LIN {X 0,Y 218.503,Z 629.529,A -85,B 0,C 180,E1 -20253.691,E2 -20253.691} C_VEL
LIN {X 0,Y 218.752,Z 627.483,A -85,B 0,C 180,E1 -20257.386,E2 -20257.386} C_VEL
LIN {X 0,Y 219.498,Z 624.035,A -85,B 0,C 180,E1 -20261.078,E2 -20261.078} C_VEL
LIN {X 0,Y 220.889,Z 619.081,A -85,B 0,C 180,E1 -20264.748,E2 -20264.748} C_VEL
LIN {X 0,Y 221.921,Z 616.025,A -85,B 0,C 180,E1 -20266.562,E2 -20266.562} C_VEL
LIN {X 0,Y 224.966,Z 612.775,A -85,B 0,C 180,E1 -20270.412,E2 -20270.412} C_VEL
LIN {X 0,Y 228.61,Z 608.967,A -85,B 0,C 180,E1 -20273.558,E2 -20273.558} C_VEL
LIN {X 0,Y 233.431,Z 603.675,A -85,B 0,C 180,E1 -20276.849,E2 -20276.849} C_VEL
LIN {X 0,Y 239.262,Z 597.121,A -85,B 0,C 180,E1 -20279.959,E2 -20279.959} C_VEL
LIN {X 0,Y 246.121,Z 589.152,A -85,B 0,C 180,E1 -20282.859,E2 -20282.859} C_VEL
LIN {X 0,Y 253.842,Z 579.668,A -85,B 0,C 180,E1 -20285.552,E2 -20285.552} C_VEL
LIN {X 0,Y 259.519,Z 572.234,A -85,B 0,C 180,E1 -20287.233,E2 -20287.233} C_VEL
LIN {X 0,Y 261.796,Z 567.859,A -85,B 0,C 180,E1 -20288.621,E2 -20288.621} C_VEL
LIN {X 0,Y 263.848,Z 563.319,A -85,B 0,C 180,E1 -20290.262,E2 -20290.262} C_VEL
LIN {X 0,Y 264.397,Z 560.907,A -85,B 0,C 180,E1 -20291.648,E2 -20291.648} C_VEL
LIN {X 0,Y 264.273,Z 558.69,A -85,B 0,C 180,E1 -20294.108,E2 -20294.108} C_VEL
LIN {X 0,Y 264.108,Z 557.741,A -85,B 0,C 180,E1 -20296.222,E2 -20296.222} C_VEL
LIN {X 0,Y 263.97,Z 557.685,A -85,B 0,C 180,E1 -20298.271,E2 -20298.271} C_VEL
LIN {X 0,Y 263.62,Z 558.789,A -85,B 0,C 180,E1 -20300.638,E2 -20300.638} C_VEL
LIN {X 0,Y 263.042,Z 560.356,A -85,B 0,C 180,E1 -20302.083,E2 -20302.083} C_VEL
LIN {X 0,Y 261.574,Z 564.149,A -85,B 0,C 180,E1 -20304.563,E2 -20304.563} C_VEL
LIN {X 0,Y 260.042,Z 567.586,A -85,B 0,C 180,E1 -20306.355,E2 -20306.355} C_VEL
LIN {X 0,Y 252.229,Z 576.861,A -85,B 0,C 180,E1 -20308.971,E2 -20308.971} C_VEL
LIN {X 0,Y 245.081,Z 584.507,A -85,B 0,C 180,E1 -20311.761,E2 -20311.761} C_VEL
LIN {X 0,Y 238.602,Z 590.64,A -85,B 0,C 180,E1 -20314.717,E2 -20314.717} C_VEL
LIN {X 0,Y 233.176,Z 595.264,A -85,B 0,C 180,E1 -20317.867,E2 -20317.867} C_VEL
LIN {X 0,Y 229.685,Z 597.919,A -85,B 0,C 180,E1 -20320.331,E2 -20320.331} C_VEL
LIN {X 0,Y 225.704,Z 600.243,A -85,B 0,C 180,E1 -20323.725,E2 -20323.725} C_VEL
LIN {X 0,Y 222.922,Z 601.265,A -85,B 0,C 180,E1 -20327.251,E2 -20327.251} C_VEL
LIN {X 0,Y 220.73,Z 600.99,A -85,B 0,C 180,E1 -20330.84,E2 -20330.84} C_VEL
LIN {X 0,Y 219.454,Z 599.351,A -85,B 0,C 180,E1 -20334.487,E2 -20334.487} C_VEL
LIN {X 0,Y 218.949,Z 596.268,A -85,B 0,C 180,E1 -20338.161,E2 -20338.161} C_VEL
LIN {X 0,Y 218.827,Z 591.637,A -85,B 0,C 180,E1 -20341.841,E2 -20341.841} C_VEL
LIN {X 0,Y 218.85,Z 586.867,A -85,B 0,C 180,E1 -20344.699,E2 -20344.699} C_VEL
LIN {X 0,Y 219.289,Z 580.046,A -85,B 0,C 180,E1 -20347.932,E2 -20347.932} C_VEL
LIN {X 0,Y 220.063,Z 571.783,A -85,B 0,C 180,E1 -20351.047,E2 -20351.047} C_VEL
LIN {X 0,Y 221.026,Z 562.858,A -85,B 0,C 180,E1 -20353.797,E2 -20353.797} C_VEL
LIN {X 0,Y 222.231,Z 554.062,A -85,B 0,C 180,E1 -20356.065,E2 -20356.065} C_VEL
LIN {X 0,Y 223.678,Z 543.655,A -85,B 0,C 180,E1 -20358.313,E2 -20358.313} C_VEL
LIN {X 0,Y 225.283,Z 531.049,A -85,B 0,C 180,E1 -20360.519,E2 -20360.519} C_VEL
LIN {X 0,Y 225.813,Z 526.308,A -85,B 0,C 180,E1 -20361.239,E2 -20361.239} C_VEL
LIN {X 0,Y 223.814,Z 512.351,A -85,B 0,C 180,E1 -20363.186,E2 -20363.186} C_VEL
LIN {X 0,Y 221.525,Z 497.373,A -85,B 0,C 180,E1 -20364.871,E2 -20364.871} C_VEL
LIN {X 0,Y 219.985,Z 485.91,A -85,B 0,C 180,E1 -20365.931,E2 -20365.931} C_VEL
LIN {X 0,Y 220.619,Z 480.954,A -85,B 0,C 180,E1 -20370.668,E2 -20370.668} C_VEL
LIN {X 0,Y 221.078,Z 477.085,A -85,B 0,C 180,E1 -20374.453,E2 -20374.453} C_VEL
LIN {X 0,Y 221.122,Z 476.819,A -85,B 0,C 180,E1 -20374.897,E2 -20374.897} C_VEL
LIN {X 0,Y 222.629,Z 479.788,A -85,B 0,C 180,E1 -20377.886,E2 -20377.886} C_VEL
LIN {X 0,Y 223.343,Z 482.152,A -85,B 0,C 180,E1 -20380.019,E2 -20380.019} C_VEL
LIN {X 0,Y 224.175,Z 486.808,A -85,B 0,C 180,E1 -20383.855,E2 -20383.855} C_VEL
LIN {X 0,Y 224.912,Z 491.35,A -85,B 0,C 180,E1 -20387.357,E2 -20387.357} C_VEL
LIN {X 0,Y 225.177,Z 493.27,A -85,B 0,C 180,E1 -20388.7,E2 -20388.7} C_VEL
LIN {X 0,Y 227.017,Z 497.219,A -85,B 0,C 180,E1 -20389.273,E2 -20389.273} C_VEL
LIN {X 0,Y 231.976,Z 510.206,A -85,B 0,C 180,E1 -20391.059,E2 -20391.059} C_VEL
LIN {X 0,Y 235.762,Z 523.157,A -85,B 0,C 180,E1 -20392.884,E2 -20392.884} C_VEL
LIN {X 0,Y 238.217,Z 535.615,A -85,B 0,C 180,E1 -20394.709,E2 -20394.709} C_VEL
LIN {X 0,Y 239.642,Z 548.301,A -85,B 0,C 180,E1 -20396.713,E2 -20396.713} C_VEL
LIN {X 0,Y 239.919,Z 556.808,A -85,B 0,C 180,E1 -20398.176,E2 -20398.176} C_VEL
LIN {X 0,Y 236.958,Z 568.177,A -85,B 0,C 180,E1 -20399.965,E2 -20399.965} C_VEL
LIN {X 0,Y 233.468,Z 579.576,A -85,B 0,C 180,E1 -20402.185,E2 -20402.185} C_VEL
LIN {X 0,Y 230.212,Z 589.775,A -85,B 0,C 180,E1 -20404.695,E2 -20404.695} C_VEL
LIN {X 0,Y 227.272,Z 598.188,A -85,B 0,C 180,E1 -20407.258,E2 -20407.258} C_VEL
LIN {X 0,Y 224.478,Z 606.213,A -85,B 0,C 180,E1 -20410.33,E2 -20410.33} C_VEL
LIN {X 0,Y 222.996,Z 610.959,A -85,B 0,C 180,E1 -20412.576,E2 -20412.576} C_VEL
LIN {X 0,Y 220.818,Z 617.133,A -85,B 0,C 180,E1 -20416.188,E2 -20416.188} C_VEL
LIN {X 0,Y 219.752,Z 620.638,A -85,B 0,C 180,E1 -20418.935,E2 -20418.935} C_VEL
LIN {X 0,Y 218.87,Z 624.059,A -85,B 0,C 180,E1 -20422.618,E2 -20422.618} C_VEL
LIN {X 0,Y 218.519,Z 626.092,A -85,B 0,C 180,E1 -20426.31,E2 -20426.31} C_VEL
LIN {X 0,Y 218.536,Z 626.788,A -85,B 0,C 180,E1 -20429.998,E2 -20429.998} C_VEL
LIN {X 0,Y 218.517,Z 626.151,A -85,B 0,C 180,E1 -20433.686,E2 -20433.686} C_VEL
LIN {X 0,Y 218.868,Z 624.168,A -85,B 0,C 180,E1 -20437.377,E2 -20437.377} C_VEL
LIN {X 0,Y 219.738,Z 620.796,A -85,B 0,C 180,E1 -20441.061,E2 -20441.061} C_VEL
LIN {X 0,Y 221.154,Z 615.933,A -85,B 0,C 180,E1 -20444.725,E2 -20444.725} C_VEL
LIN {X 0,Y 222.932,Z 611.22,A -85,B 0,C 180,E1 -20447.424,E2 -20447.424} C_VEL
LIN {X 0,Y 225.05,Z 604.615,A -85,B 0,C 180,E1 -20450.469,E2 -20450.469} C_VEL
LIN {X 0,Y 228.117,Z 595.91,A -85,B 0,C 180,E1 -20453.608,E2 -20453.608} C_VEL
LIN {X 0,Y 231.148,Z 587.038,A -85,B 0,C 180,E1 -20456.157,E2 -20456.157} C_VEL
LIN {X 0,Y 234.623,Z 576.293,A -85,B 0,C 180,E1 -20458.635,E2 -20458.635} C_VEL
LIN {X 0,Y 237.684,Z 565.995,A -85,B 0,C 180,E1 -20460.535,E2 -20460.535} C_VEL
LIN {X 0,Y 240.047,Z 556.241,A -85,B 0,C 180,E1 -20462.044,E2 -20462.044} C_VEL
LIN {X 0,Y 239.422,Z 545.365,A -85,B 0,C 180,E1 -20463.896,E2 -20463.896} C_VEL
LIN {X 0,Y 237.78,Z 532.647,A -85,B 0,C 180,E1 -20465.861,E2 -20465.861} C_VEL
LIN {X 0,Y 234.898,Z 519.812,A -85,B 0,C 180,E1 -20467.73,E2 -20467.73} C_VEL
LIN {X 0,Y 230.885,Z 507.056,A -85,B 0,C 180,E1 -20469.517,E2 -20469.517} C_VEL
LIN {X 0,Y 226.816,Z 496.9,A -85,B 0,C 180,E1 -20470.939,E2 -20470.939} C_VEL
LIN {X 0,Y 225.184,Z 493.126,A -85,B 0,C 180,E1 -20471.492,E2 -20471.492} C_VEL
LIN {X 0,Y 224.486,Z 488.194,A -85,B 0,C 180,E1 -20475.219,E2 -20475.219} C_VEL
LIN {X 0,Y 223.668,Z 483.614,A -85,B 0,C 180,E1 -20478.944,E2 -20478.944} C_VEL
LIN {X 0,Y 222.607,Z 478.78,A -85,B 0,C 180,E1 -20483.14,E2 -20483.14} C_VEL
LIN {X 0,Y 221.548,Z 474.367,A -85,B 0,C 180,E1 -20487.365,E2 -20487.365} C_VEL
LIN {X 0,Y 220.874,Z 471.591,A -85,B 0,C 180,E1 -20490.187,E2 -20490.187} C_VEL
LIN {X 0,Y 220.888,Z 471.58,A -85,B 0,C 180,E1 -20493.548,E2 -20493.548} C_VEL
LIN {X 0,Y 220.927,Z 471.571,A -85,B 0,C 180,E1 -20497.558,E2 -20497.558} C_VEL
LIN {X 0,Y 220.984,Z 471.579,A -85,B 0,C 180,E1 -20502.563,E2 -20502.563} C_VEL
LIN {X 0,Y 221.017,Z 471.578,A -85,B 0,C 180,E1 -20507.139,E2 -20507.139} C_VEL
LIN {X 0,Y 221.248,Z 471.545,A -85,B 0,C 180,E1 -20510.861,E2 -20510.861} C_VEL
LIN {X 0,Y 221.303,Z 471.543,A -85,B 0,C 180,E1 -20512.702,E2 -20512.702} C_VEL
LIN {X 0,Y 221.513,Z 471.51,A -85,B 0,C 180,E1 -20518.182,E2 -20518.182} C_VEL
LIN {X 0,Y 221.503,Z 471.499,A -85,B 0,C 180,E1 -20521.818,E2 -20521.818} C_VEL
LIN {X 0,Y 221.301,Z 471.545,A -85,B 0,C 180,E1 -20527.298,E2 -20527.298} C_VEL
LIN {X 0,Y 221.108,Z 471.535,A -85,B 0,C 180,E1 -20530.994,E2 -20530.994} C_VEL
LIN {X 0,Y 221.007,Z 471.553,A -85,B 0,C 180,E1 -20536.63,E2 -20536.63} C_VEL
LIN {X 0,Y 220.883,Z 471.597,A -85,B 0,C 180,E1 -20540.487,E2 -20540.487} C_VEL
LIN {X 0,Y 220.858,Z 471.597,A -85,B 0,C 180,E1 -20544.436,E2 -20544.436} C_VEL
LIN {X 0,Y 220.828,Z 471.599,A -85,B 0,C 180,E1 -20548.515,E2 -20548.515} C_VEL
LIN {X 0,Y 220.816,Z 471.606,A -85,B 0,C 180,E1 -20552.756,E2 -20552.756} C_VEL
LIN {X 0,Y 220.835,Z 471.618,A -85,B 0,C 180,E1 -20557.814,E2 -20557.814} C_VEL
LIN {X 0,Y 222.87,Z 477.355,A -85,B 0,C 180,E1 -20561.469,E2 -20561.469} C_VEL
LIN {X 0,Y 224.638,Z 484.826,A -85,B 0,C 180,E1 -20565.377,E2 -20565.377} C_VEL
LIN {X 0,Y 226.301,Z 492.458,A -85,B 0,C 180,E1 -20568.941,E2 -20568.941} C_VEL
LIN {X 0,Y 233.494,Z 506.389,A -85,B 0,C 180,E1 -20571.066,E2 -20571.066} C_VEL
LIN {X 0,Y 233.812,Z 507.056,A -85,B 0,C 180,E1 -20571.165,E2 -20571.165} C_VEL
LIN {X 0,Y 235,Z 510.338,A -85,B 0,C 180,E1 -20571.596,E2 -20571.596} C_VEL
LIN {X 0,Y 235.618,Z 515.851,A -85,B 0,C 180,E1 -20572.088,E2 -20572.088} C_VEL
LIN {X 0,Y 235.189,Z 521.596,A -85,B 0,C 180,E1 -20572.474,E2 -20572.474} C_VEL
LIN {X 0,Y 233.665,Z 531.413,A -85,B 0,C 180,E1 -20573.154,E2 -20573.154} C_VEL
LIN {X 0,Y 233.415,Z 536.957,A -85,B 0,C 180,E1 -20573.756,E2 -20573.756} C_VEL
LIN {X 0,Y 233.847,Z 550.482,A -85,B 0,C 180,E1 -20575.704,E2 -20575.704} C_VEL
LIN {X 0,Y 233.66,Z 558.252,A -85,B 0,C 180,E1 -20576.967,E2 -20576.967} C_VEL
LIN {X 0,Y 230.585,Z 570.015,A -85,B 0,C 180,E1 -20578.795,E2 -20578.795} C_VEL
LIN {X 0,Y 227.354,Z 580.759,A -85,B 0,C 180,E1 -20580.868,E2 -20580.868} C_VEL
LIN {X 0,Y 223.723,Z 591.371,A -85,B 0,C 180,E1 -20583.41,E2 -20583.41} C_VEL
LIN {X 0,Y 220.653,Z 600.117,A -85,B 0,C 180,E1 -20586.043,E2 -20586.043} C_VEL
LIN {X 0,Y 217.61,Z 608.489,A -85,B 0,C 180,E1 -20589.193,E2 -20589.193} C_VEL
LIN {X 0,Y 215.618,Z 614.309,A -85,B 0,C 180,E1 -20591.965,E2 -20591.965} C_VEL
LIN {X 0,Y 214.015,Z 619.098,A -85,B 0,C 180,E1 -20594.772,E2 -20594.772} C_VEL
LIN {X 0,Y 212.481,Z 624.036,A -85,B 0,C 180,E1 -20598.556,E2 -20598.556} C_VEL
LIN {X 0,Y 211.675,Z 627.468,A -85,B 0,C 180,E1 -20602.371,E2 -20602.371} C_VEL
LIN {X 0,Y 211.416,Z 629.495,A -85,B 0,C 180,E1 -20606.19,E2 -20606.19} C_VEL
LIN {X 0,Y 211.455,Z 630.163,A -85,B 0,C 180,E1 -20610.002,E2 -20610.002} C_VEL
LIN {X 0,Y 211.417,Z 629.473,A -85,B 0,C 180,E1 -20613.814,E2 -20613.814} C_VEL
LIN {X 0,Y 211.677,Z 627.427,A -85,B 0,C 180,E1 -20617.634,E2 -20617.634} C_VEL
LIN {X 0,Y 212.48,Z 623.978,A -85,B 0,C 180,E1 -20621.449,E2 -20621.449} C_VEL
LIN {X 0,Y 214.011,Z 619.025,A -85,B 0,C 180,E1 -20625.234,E2 -20625.234} C_VEL
LIN {X 0,Y 215.073,Z 616.044,A -85,B 0,C 180,E1 -20627.106,E2 -20627.106} C_VEL
LIN {X 0,Y 218.11,Z 613.291,A -85,B 0,C 180,E1 -20630.861,E2 -20630.861} C_VEL
LIN {X 0,Y 222.157,Z 609.591,A -85,B 0,C 180,E1 -20634.286,E2 -20634.286} C_VEL
LIN {X 0,Y 227.184,Z 604.681,A -85,B 0,C 180,E1 -20637.65,E2 -20637.65} C_VEL
LIN {X 0,Y 233.28,Z 598.565,A -85,B 0,C 180,E1 -20640.81,E2 -20640.81} C_VEL
LIN {X 0,Y 240.399,Z 591.12,A -85,B 0,C 180,E1 -20643.745,E2 -20643.745} C_VEL
LIN {X 0,Y 248.381,Z 582.202,A -85,B 0,C 180,E1 -20646.458,E2 -20646.458} C_VEL
LIN {X 0,Y 254.785,Z 574.607,A -85,B 0,C 180,E1 -20648.299,E2 -20648.299} C_VEL
LIN {X 0,Y 256.737,Z 571.335,A -85,B 0,C 180,E1 -20649.402,E2 -20649.402} C_VEL
LIN {X 0,Y 258.593,Z 567.913,A -85,B 0,C 180,E1 -20650.715,E2 -20650.715} C_VEL
LIN {X 0,Y 259.308,Z 565.951,A -85,B 0,C 180,E1 -20651.81,E2 -20651.81} C_VEL
LIN {X 0,Y 259.388,Z 564.759,A -85,B 0,C 180,E1 -20652.983,E2 -20652.983} C_VEL
LIN {X 0,Y 259.281,Z 563.344,A -85,B 0,C 180,E1 -20655.191,E2 -20655.191} C_VEL
LIN {X 0,Y 259.133,Z 562.835,A -85,B 0,C 180,E1 -20657.31,E2 -20657.31} C_VEL
LIN {X 0,Y 258.797,Z 563.312,A -85,B 0,C 180,E1 -20659.5,E2 -20659.5} C_VEL
LIN {X 0,Y 258.229,Z 564.598,A -85,B 0,C 180,E1 -20661.247,E2 -20661.247} C_VEL
LIN {X 0,Y 257.123,Z 566.844,A -85,B 0,C 180,E1 -20663.035,E2 -20663.035} C_VEL
LIN {X 0,Y 255.728,Z 569.568,A -85,B 0,C 180,E1 -20664.751,E2 -20664.751} C_VEL
LIN {X 0,Y 254.808,Z 571.133,A -85,B 0,C 180,E1 -20665.568,E2 -20665.568} C_VEL
LIN {X 0,Y 246.576,Z 579.858,A -85,B 0,C 180,E1 -20668.177,E2 -20668.177} C_VEL
LIN {X 0,Y 239.146,Z 586.889,A -85,B 0,C 180,E1 -20670.994,E2 -20670.994} C_VEL
LIN {X 0,Y 232.439,Z 592.557,A -85,B 0,C 180,E1 -20673.997,E2 -20673.997} C_VEL
LIN {X 0,Y 228.115,Z 595.859,A -85,B 0,C 180,E1 -20676.39,E2 -20676.39} C_VEL
LIN {X 0,Y 223.119,Z 599.111,A -85,B 0,C 180,E1 -20679.727,E2 -20679.727} C_VEL
LIN {X 0,Y 218.953,Z 601.142,A -85,B 0,C 180,E1 -20683.209,E2 -20683.209} C_VEL
LIN {X 0,Y 216.03,Z 601.851,A -85,B 0,C 180,E1 -20686.837,E2 -20686.837} C_VEL
LIN {X 0,Y 213.626,Z 601.177,A -85,B 0,C 180,E1 -20690.747,E2 -20690.747} C_VEL
LIN {X 0,Y 212.388,Z 599.301,A -85,B 0,C 180,E1 -20694.303,E2 -20694.303} C_VEL
LIN {X 0,Y 211.885,Z 595.957,A -85,B 0,C 180,E1 -20698.099,E2 -20698.099} C_VEL
LIN {X 0,Y 211.749,Z 592.444,A -85,B 0,C 180,E1 -20700.951,E2 -20700.951} C_VEL
LIN {X 0,Y 211.774,Z 587.955,A -85,B 0,C 180,E1 -20703.806,E2 -20703.806} C_VEL
LIN {X 0,Y 212.095,Z 581.373,A -85,B 0,C 180,E1 -20707.138,E2 -20707.138} C_VEL
LIN {X 0,Y 212.808,Z 573.165,A -85,B 0,C 180,E1 -20710.465,E2 -20710.465} C_VEL
LIN {X 0,Y 213.731,Z 564.419,A -85,B 0,C 180,E1 -20713.308,E2 -20713.308} C_VEL
LIN {X 0,Y 215.138,Z 553.94,A -85,B 0,C 180,E1 -20716.122,E2 -20716.122} C_VEL
LIN {X 0,Y 216.763,Z 542.287,A -85,B 0,C 180,E1 -20718.674,E2 -20718.674} C_VEL
LIN {X 0,Y 218.447,Z 529.333,A -85,B 0,C 180,E1 -20720.982,E2 -20720.982} C_VEL
LIN {X 0,Y 218.682,Z 526.244,A -85,B 0,C 180,E1 -20721.459,E2 -20721.459} C_VEL
LIN {X 0,Y 216.74,Z 512.928,A -85,B 0,C 180,E1 -20723.378,E2 -20723.378} C_VEL
LIN {X 0,Y 214.476,Z 497.918,A -85,B 0,C 180,E1 -20725.124,E2 -20725.124} C_VEL
LIN {X 0,Y 212.964,Z 486.1,A -85,B 0,C 180,E1 -20726.268,E2 -20726.268} C_VEL
LIN {X 0,Y 213.387,Z 482.689,A -85,B 0,C 180,E1 -20729.606,E2 -20729.606} C_VEL
LIN {X 0,Y 213.954,Z 478.47,A -85,B 0,C 180,E1 -20733.876,E2 -20733.876} C_VEL
LIN {X 0,Y 215.61,Z 481.474,A -85,B 0,C 180,E1 -20737.087,E2 -20737.087} C_VEL
LIN {X 0,Y 216.329,Z 483.177,A -85,B 0,C 180,E1 -20738.764,E2 -20738.764} C_VEL
LIN {X 0,Y 217.226,Z 487.854,A -85,B 0,C 180,E1 -20742.799,E2 -20742.799} C_VEL
LIN {X 0,Y 218.133,Z 493.23,A -85,B 0,C 180,E1 -20747.054,E2 -20747.054} C_VEL
LIN {X 0,Y 219.817,Z 496.81,A -85,B 0,C 180,E1 -20747.62,E2 -20747.62} C_VEL
LIN {X 0,Y 220.987,Z 498.779,A -85,B 0,C 180,E1 -20747.994,E2 -20747.994} C_VEL
LIN {X 0,Y 224.109,Z 506.194,A -85,B 0,C 180,E1 -20749.137,E2 -20749.137} C_VEL
LIN {X 0,Y 227.4,Z 516.028,A -85,B 0,C 180,E1 -20750.593,E2 -20750.593} C_VEL
LIN {X 0,Y 230.522,Z 528.189,A -85,B 0,C 180,E1 -20752.436,E2 -20752.436} C_VEL
LIN {X 0,Y 232.621,Z 540.957,A -85,B 0,C 180,E1 -20754.453,E2 -20754.453} C_VEL
LIN {X 0,Y 233.594,Z 553.147,A -85,B 0,C 180,E1 -20756.54,E2 -20756.54} C_VEL
LIN {X 0,Y 233.672,Z 557.651,A -85,B 0,C 180,E1 -20757.367,E2 -20757.367} C_VEL
LIN {X 0,Y 230.503,Z 569.379,A -85,B 0,C 180,E1 -20759.287,E2 -20759.287} C_VEL
LIN {X 0,Y 227.214,Z 579.627,A -85,B 0,C 180,E1 -20761.349,E2 -20761.349} C_VEL
LIN {X 0,Y 223.798,Z 589.828,A -85,B 0,C 180,E1 -20763.916,E2 -20763.916} C_VEL
LIN {X 0,Y 220.72,Z 598.242,A -85,B 0,C 180,E1 -20766.544,E2 -20766.544} C_VEL
LIN {X 0,Y 217.894,Z 605.846,A -85,B 0,C 180,E1 -20769.502,E2 -20769.502} C_VEL
LIN {X 0,Y 216.205,Z 611.015,A -85,B 0,C 180,E1 -20772.01,E2 -20772.01} C_VEL
LIN {X 0,Y 213.902,Z 617.189,A -85,B 0,C 180,E1 -20775.732,E2 -20775.732} C_VEL
LIN {X 0,Y 212.765,Z 620.695,A -85,B 0,C 180,E1 -20778.567,E2 -20778.567} C_VEL
LIN {X 0,Y 211.83,Z 624.115,A -85,B 0,C 180,E1 -20782.371,E2 -20782.371} C_VEL
LIN {X 0,Y 211.438,Z 626.148,A -85,B 0,C 180,E1 -20786.186,E2 -20786.186} C_VEL
LIN {X 0,Y 211.438,Z 626.844,A -85,B 0,C 180,E1 -20789.998,E2 -20789.998} C_VEL
LIN {X 0,Y 211.437,Z 626.207,A -85,B 0,C 180,E1 -20793.809,E2 -20793.809} C_VEL
LIN {X 0,Y 211.827,Z 624.223,A -85,B 0,C 180,E1 -20797.624,E2 -20797.624} C_VEL
LIN {X 0,Y 212.749,Z 620.85,A -85,B 0,C 180,E1 -20801.429,E2 -20801.429} C_VEL
LIN {X 0,Y 214.27,Z 615.987,A -85,B 0,C 180,E1 -20805.21,E2 -20805.21} C_VEL
LIN {X 0,Y 216.136,Z 611.273,A -85,B 0,C 180,E1 -20807.991,E2 -20807.991} C_VEL
LIN {X 0,Y 218.196,Z 605.162,A -85,B 0,C 180,E1 -20810.92,E2 -20810.92} C_VEL
LIN {X 0,Y 221.114,Z 597.295,A -85,B 0,C 180,E1 -20813.904,E2 -20813.904} C_VEL
LIN {X 0,Y 224.232,Z 588.689,A -85,B 0,C 180,E1 -20816.525,E2 -20816.525} C_VEL
LIN {X 0,Y 227.766,Z 578.258,A -85,B 0,C 180,E1 -20819.074,E2 -20819.074} C_VEL
LIN {X 0,Y 231.061,Z 567.733,A -85,B 0,C 180,E1 -20821.133,E2 -20821.133} C_VEL
LIN {X 0,Y 233.734,Z 557.654,A -85,B 0,C 180,E1 -20822.765,E2 -20822.765} C_VEL
LIN {X 0,Y 233.138,Z 545.396,A -85,B 0,C 180,E1 -20824.94,E2 -20824.94} C_VEL
LIN {X 0,Y 231.594,Z 533.513,A -85,B 0,C 180,E1 -20826.87,E2 -20826.87} C_VEL
LIN {X 0,Y 229.039,Z 521.723,A -85,B 0,C 180,E1 -20828.689,E2 -20828.689} C_VEL
LIN {X 0,Y 225.106,Z 508.715,A -85,B 0,C 180,E1 -20830.625,E2 -20830.625} C_VEL
LIN {X 0,Y 221.674,Z 500.227,A -85,B 0,C 180,E1 -20831.926,E2 -20831.926} C_VEL
LIN {X 0,Y 219.887,Z 496.817,A -85,B 0,C 180,E1 -20832.524,E2 -20832.524} C_VEL
LIN {X 0,Y 218.165,Z 493.1,A -85,B 0,C 180,E1 -20833.148,E2 -20833.148} C_VEL
LIN {X 0,Y 217.349,Z 488.069,A -85,B 0,C 180,E1 -20837.231,E2 -20837.231} C_VEL
LIN {X 0,Y 216.293,Z 482.673,A -85,B 0,C 180,E1 -20841.876,E2 -20841.876} C_VEL
LIN {X 0,Y 215.645,Z 479.835,A -85,B 0,C 180,E1 -20844.559,E2 -20844.559} C_VEL
LIN {X 0,Y 214.385,Z 474.964,A -85,B 0,C 180,E1 -20849.461,E2 -20849.461} C_VEL
LIN {X 0,Y 213.808,Z 472.465,A -85,B 0,C 180,E1 -20852.362,E2 -20852.362} C_VEL
LIN {X 0,Y 213.858,Z 472.455,A -85,B 0,C 180,E1 -20856.942,E2 -20856.942} C_VEL
LIN {X 0,Y 213.961,Z 472.455,A -85,B 0,C 180,E1 -20862.805,E2 -20862.805} C_VEL
LIN {X 0,Y 213.972,Z 472.458,A -85,B 0,C 180,E1 -20866.708,E2 -20866.708} C_VEL
LIN {X 0,Y 214.187,Z 472.427,A -85,B 0,C 180,E1 -20870.557,E2 -20870.557} C_VEL
LIN {X 0,Y 214.239,Z 472.42,A -85,B 0,C 180,E1 -20872.46,E2 -20872.46} C_VEL
LIN {X 0,Y 214.47,Z 472.388,A -85,B 0,C 180,E1 -20878.122,E2 -20878.122} C_VEL
LIN {X 0,Y 214.545,Z 472.387,A -85,B 0,C 180,E1 -20880,E2 -20880} C_VEL
LIN {X 0,Y 214.437,Z 472.378,A -85,B 0,C 180,E1 -20881.878,E2 -20881.878} C_VEL
LIN {X 0,Y 214.238,Z 472.424,A -85,B 0,C 180,E1 -20887.54,E2 -20887.54} C_VEL
LIN {X 0,Y 214.04,Z 472.417,A -85,B 0,C 180,E1 -20891.362,E2 -20891.362} C_VEL
LIN {X 0,Y 213.933,Z 472.451,A -85,B 0,C 180,E1 -20895.237,E2 -20895.237} C_VEL
LIN {X 0,Y 213.83,Z 472.456,A -85,B 0,C 180,E1 -20899.188,E2 -20899.188} C_VEL
LIN {X 0,Y 213.838,Z 472.472,A -85,B 0,C 180,E1 -20903.228,E2 -20903.228} C_VEL
LIN {X 0,Y 213.82,Z 472.474,A -85,B 0,C 180,E1 -20907.451,E2 -20907.451} C_VEL
LIN {X 0,Y 213.771,Z 472.48,A -85,B 0,C 180,E1 -20911.737,E2 -20911.737} C_VEL
LIN {X 0,Y 213.76,Z 472.506,A -85,B 0,C 180,E1 -20915.419,E2 -20915.419} C_VEL
LIN {X 0,Y 215.78,Z 478.094,A -85,B 0,C 180,E1 -20919.428,E2 -20919.428} C_VEL
LIN {X 0,Y 217.125,Z 482.011,A -85,B 0,C 180,E1 -20921.89,E2 -20921.89} C_VEL
LIN {X 0,Y 218.849,Z 490.276,A -85,B 0,C 180,E1 -20926.266,E2 -20926.266} C_VEL
LIN {X 0,Y 219.422,Z 492.69,A -85,B 0,C 180,E1 -20927.362,E2 -20927.362} C_VEL
LIN {X 0,Y 226.868,Z 506.825,A -85,B 0,C 180,E1 -20929.722,E2 -20929.722} C_VEL
LIN {X 0,Y 229.838,Z 513.766,A -85,B 0,C 180,E1 -20930.799,E2 -20930.799} C_VEL
LIN {X 0,Y 232.425,Z 526.583,A -85,B 0,C 180,E1 -20932.411,E2 -20932.411} C_VEL
LIN {X 0,Y 233.415,Z 536.957,A -85,B 0,C 180,E1 -20933.756,E2 -20933.756} C_VEL
LIN {X 0,Y 233.216,Z 542.264,A -85,B 0,C 180,E1 -20934.399,E2 -20934.399} C_VEL
LIN {X 0,Y 232.056,Z 547.638,A -85,B 0,C 180,E1 -20934.963,E2 -20934.963} C_VEL
LIN {X 0,Y 228.326,Z 558.167,A -85,B 0,C 180,E1 -20936.079,E2 -20936.079} C_VEL
LIN {X 0,Y 225.978,Z 564.918,A -85,B 0,C 180,E1 -20937.006,E2 -20937.006} C_VEL
LIN {X 0,Y 222.511,Z 576.659,A -85,B 0,C 180,E1 -20939.122,E2 -20939.122} C_VEL
LIN {X 0,Y 219.191,Z 586.283,A -85,B 0,C 180,E1 -20941.255,E2 -20941.255} C_VEL
LIN {X 0,Y 215.706,Z 595.9,A -85,B 0,C 180,E1 -20943.909,E2 -20943.909} C_VEL
LIN {X 0,Y 212.667,Z 603.864,A -85,B 0,C 180,E1 -20946.639,E2 -20946.639} C_VEL
LIN {X 0,Y 210.102,Z 610.578,A -85,B 0,C 180,E1 -20949.49,E2 -20949.49} C_VEL
LIN {X 0,Y 208.236,Z 615.967,A -85,B 0,C 180,E1 -20952.32,E2 -20952.32} C_VEL
LIN {X 0,Y 206.154,Z 621.709,A -85,B 0,C 180,E1 -20956.197,E2 -20956.197} C_VEL
LIN {X 0,Y 204.97,Z 625.878,A -85,B 0,C 180,E1 -20960.131,E2 -20960.131} C_VEL
LIN {X 0,Y 204.4,Z 628.597,A -85,B 0,C 180,E1 -20964.082,E2 -20964.082} C_VEL
LIN {X 0,Y 204.322,Z 629.943,A -85,B 0,C 180,E1 -20968.031,E2 -20968.031} C_VEL
LIN {X 0,Y 204.359,Z 630.107,A -85,B 0,C 180,E1 -20970.002,E2 -20970.002} C_VEL
LIN {X 0,Y 204.336,Z 629.417,A -85,B 0,C 180,E1 -20973.947,E2 -20973.947} C_VEL
LIN {X 0,Y 204.628,Z 627.371,A -85,B 0,C 180,E1 -20977.899,E2 -20977.899} C_VEL
LIN {X 0,Y 205.483,Z 623.922,A -85,B 0,C 180,E1 -20981.844,E2 -20981.844} C_VEL
LIN {X 0,Y 207.122,Z 618.969,A -85,B 0,C 180,E1 -20985.753,E2 -20985.753} C_VEL
LIN {X 0,Y 208.25,Z 615.975,A -85,B 0,C 180,E1 -20987.684,E2 -20987.684} C_VEL
LIN {X 0,Y 211.389,Z 613.629,A -85,B 0,C 180,E1 -20991.454,E2 -20991.454} C_VEL
LIN {X 0,Y 215.724,Z 610.197,A -85,B 0,C 180,E1 -20995.06,E2 -20995.06} C_VEL
LIN {X 0,Y 220.987,Z 605.667,A -85,B 0,C 180,E1 -20998.495,E2 -20998.495} C_VEL
LIN {X 0,Y 227.344,Z 599.971,A -85,B 0,C 180,E1 -21001.706,E2 -21001.706} C_VEL
LIN {X 0,Y 234.719,Z 593,A -85,B 0,C 180,E1 -21004.676,E2 -21004.676} C_VEL
LIN {X 0,Y 242.958,Z 584.671,A -85,B 0,C 180,E1 -21007.409,E2 -21007.409} C_VEL
LIN {X 0,Y 249.705,Z 577.415,A -85,B 0,C 180,E1 -21009.294,E2 -21009.294} C_VEL
LIN {X 0,Y 251.344,Z 575.187,A -85,B 0,C 180,E1 -21010.027,E2 -21010.027} C_VEL
LIN {X 0,Y 253.694,Z 571.372,A -85,B 0,C 180,E1 -21011.674,E2 -21011.674} C_VEL
LIN {X 0,Y 254.237,Z 569.715,A -85,B 0,C 180,E1 -21013.004,E2 -21013.004} C_VEL
LIN {X 0,Y 254.14,Z 568.115,A -85,B 0,C 180,E1 -21015.975,E2 -21015.975} C_VEL
LIN {X 0,Y 253.843,Z 568.012,A -85,B 0,C 180,E1 -21018.379,E2 -21018.379} C_VEL
LIN {X 0,Y 253.297,Z 568.872,A -85,B 0,C 180,E1 -21020.345,E2 -21020.345} C_VEL
LIN {X 0,Y 253.001,Z 569.415,A -85,B 0,C 180,E1 -21021.062,E2 -21021.062} C_VEL
LIN {X 0,Y 251.455,Z 571.839,A -85,B 0,C 180,E1 -21023.065,E2 -21023.065} C_VEL
LIN {X 0,Y 250.643,Z 573.113,A -85,B 0,C 180,E1 -21023.926,E2 -21023.926} C_VEL
LIN {X 0,Y 249.41,Z 574.656,A -85,B 0,C 180,E1 -21024.714,E2 -21024.714} C_VEL
LIN {X 0,Y 240.935,Z 582.721,A -85,B 0,C 180,E1 -21027.341,E2 -21027.341} C_VEL
LIN {X 0,Y 233.246,Z 589.281,A -85,B 0,C 180,E1 -21030.187,E2 -21030.187} C_VEL
LIN {X 0,Y 226.292,Z 594.442,A -85,B 0,C 180,E1 -21033.235,E2 -21033.235} C_VEL
LIN {X 0,Y 221.785,Z 597.439,A -85,B 0,C 180,E1 -21035.673,E2 -21035.673} C_VEL
LIN {X 0,Y 216.573,Z 600.32,A -85,B 0,C 180,E1 -21039.087,E2 -21039.087} C_VEL
LIN {X 0,Y 212.213,Z 601.956,A -85,B 0,C 180,E1 -21042.659,E2 -21042.659} C_VEL
LIN {X 0,Y 209.134,Z 602.323,A -85,B 0,C 180,E1 -21046.395,E2 -21046.395} C_VEL
LIN {X 0,Y 206.743,Z 601.427,A -85,B 0,C 180,E1 -21050.214,E2 -21050.214} C_VEL
LIN {X 0,Y 205.328,Z 599.21,A -85,B 0,C 180,E1 -21054.106,E2 -21054.106} C_VEL
LIN {X 0,Y 204.822,Z 595.579,A -85,B 0,C 180,E1 -21058.034,E2 -21058.034} C_VEL
LIN {X 0,Y 204.701,Z 590.39,A -85,B 0,C 180,E1 -21061.968,E2 -21061.968} C_VEL
LIN {X 0,Y 204.787,Z 584.643,A -85,B 0,C 180,E1 -21065.283,E2 -21065.283} C_VEL
LIN {X 0,Y 205.221,Z 577.992,A -85,B 0,C 180,E1 -21068.369,E2 -21068.369} C_VEL
LIN {X 0,Y 206.138,Z 568.865,A -85,B 0,C 180,E1 -21071.804,E2 -21071.804} C_VEL
LIN {X 0,Y 207.247,Z 559.316,A -85,B 0,C 180,E1 -21074.734,E2 -21074.734} C_VEL
LIN {X 0,Y 208.694,Z 548.749,A -85,B 0,C 180,E1 -21077.39,E2 -21077.39} C_VEL
LIN {X 0,Y 210.291,Z 537.131,A -85,B 0,C 180,E1 -21079.778,E2 -21079.778} C_VEL
LIN {X 0,Y 211.601,Z 526.715,A -85,B 0,C 180,E1 -21081.564,E2 -21081.564} C_VEL
LIN {X 0,Y 209.671,Z 513.292,A -85,B 0,C 180,E1 -21083.574,E2 -21083.574} C_VEL
LIN {X 0,Y 207.333,Z 497.723,A -85,B 0,C 180,E1 -21085.454,E2 -21085.454} C_VEL
LIN {X 0,Y 205.922,Z 486.294,A -85,B 0,C 180,E1 -21086.579,E2 -21086.579} C_VEL
LIN {X 0,Y 206.461,Z 482.208,A -85,B 0,C 180,E1 -21090.704,E2 -21090.704} C_VEL
LIN {X 0,Y 206.803,Z 480.258,A -85,B 0,C 180,E1 -21092.842,E2 -21092.842} C_VEL
LIN {X 0,Y 208.455,Z 482.967,A -85,B 0,C 180,E1 -21095.984,E2 -21095.984} C_VEL
LIN {X 0,Y 209.536,Z 485.256,A -85,B 0,C 180,E1 -21098.353,E2 -21098.353} C_VEL
LIN {X 0,Y 210.36,Z 489.218,A -85,B 0,C 180,E1 -21101.928,E2 -21101.928} C_VEL
LIN {X 0,Y 211.025,Z 493.243,A -85,B 0,C 180,E1 -21105.234,E2 -21105.234} C_VEL
LIN {X 0,Y 212.782,Z 496.77,A -85,B 0,C 180,E1 -21105.867,E2 -21105.867} C_VEL
LIN {X 0,Y 214.096,Z 498.788,A -85,B 0,C 180,E1 -21106.313,E2 -21106.313} C_VEL
LIN {X 0,Y 217.635,Z 505.845,A -85,B 0,C 180,E1 -21107.62,E2 -21107.62} C_VEL
LIN {X 0,Y 221.68,Z 517.961,A -85,B 0,C 180,E1 -21109.542,E2 -21109.542} C_VEL
LIN {X 0,Y 224.627,Z 529.882,A -85,B 0,C 180,E1 -21111.462,E2 -21111.462} C_VEL
LIN {X 0,Y 226.501,Z 542.008,A -85,B 0,C 180,E1 -21113.484,E2 -21113.484} C_VEL
LIN {X 0,Y 227.343,Z 553.597,A -85,B 0,C 180,E1 -21115.563,E2 -21115.563} C_VEL
LIN {X 0,Y 227.398,Z 558.811,A -85,B 0,C 180,E1 -21116.561,E2 -21116.561} C_VEL
LIN {X 0,Y 224.094,Z 570.573,A -85,B 0,C 180,E1 -21118.572,E2 -21118.572} C_VEL
LIN {X 0,Y 220.346,Z 581.526,A -85,B 0,C 180,E1 -21120.893,E2 -21120.893} C_VEL
LIN {X 0,Y 216.847,Z 591.361,A -85,B 0,C 180,E1 -21123.534,E2 -21123.534} C_VEL
LIN {X 0,Y 213.21,Z 600.738,A -85,B 0,C 180,E1 -21126.697,E2 -21126.697} C_VEL
LIN {X 0,Y 210.685,Z 607.375,A -85,B 0,C 180,E1 -21129.524,E2 -21129.524} C_VEL
LIN {X 0,Y 208.741,Z 612.778,A -85,B 0,C 180,E1 -21132.359,E2 -21132.359} C_VEL
LIN {X 0,Y 206.981,Z 617.246,A -85,B 0,C 180,E1 -21135.244,E2 -21135.244} C_VEL
LIN {X 0,Y 205.795,Z 620.751,A -85,B 0,C 180,E1 -21138.174,E2 -21138.174} C_VEL
LIN {X 0,Y 204.769,Z 624.171,A -85,B 0,C 180,E1 -21142.107,E2 -21142.107} C_VEL
LIN {X 0,Y 204.34,Z 626.204,A -85,B 0,C 180,E1 -21146.053,E2 -21146.053} C_VEL
LIN {X 0,Y 204.342,Z 626.899,A -85,B 0,C 180,E1 -21149.998,E2 -21149.998} C_VEL
LIN {X 0,Y 204.339,Z 626.262,A -85,B 0,C 180,E1 -21153.942,E2 -21153.942} C_VEL
LIN {X 0,Y 204.766,Z 624.278,A -85,B 0,C 180,E1 -21157.888,E2 -21157.888} C_VEL
LIN {X 0,Y 205.777,Z 620.905,A -85,B 0,C 180,E1 -21161.822,E2 -21161.822} C_VEL
LIN {X 0,Y 207.409,Z 616.04,A -85,B 0,C 180,E1 -21165.726,E2 -21165.726} C_VEL
LIN {X 0,Y 209.36,Z 611.325,A -85,B 0,C 180,E1 -21168.594,E2 -21168.594} C_VEL
LIN {X 0,Y 211.831,Z 604.495,A -85,B 0,C 180,E1 -21171.913,E2 -21171.913} C_VEL
LIN {X 0,Y 215.162,Z 596.009,A -85,B 0,C 180,E1 -21175.124,E2 -21175.124} C_VEL
LIN {X 0,Y 218.473,Z 587.133,A -85,B 0,C 180,E1 -21177.801,E2 -21177.801} C_VEL
LIN {X 0,Y 222.251,Z 576.381,A -85,B 0,C 180,E1 -21180.391,E2 -21180.391} C_VEL
LIN {X 0,Y 225.872,Z 564.998,A -85,B 0,C 180,E1 -21182.56,E2 -21182.56} C_VEL
LIN {X 0,Y 227.454,Z 559.041,A -85,B 0,C 180,E1 -21183.531,E2 -21183.531} C_VEL
LIN {X 0,Y 227.101,Z 548.027,A -85,B 0,C 180,E1 -21185.598,E2 -21185.598} C_VEL
LIN {X 0,Y 225.729,Z 535.792,A -85,B 0,C 180,E1 -21187.704,E2 -21187.704} C_VEL
LIN {X 0,Y 223.408,Z 524.378,A -85,B 0,C 180,E1 -21189.579,E2 -21189.579} C_VEL
LIN {X 0,Y 219.924,Z 512.106,A -85,B 0,C 180,E1 -21191.529,E2 -21191.529} C_VEL
LIN {X 0,Y 216.936,Z 504.328,A -85,B 0,C 180,E1 -21192.82,E2 -21192.82} C_VEL
LIN {X 0,Y 213.321,Z 497.423,A -85,B 0,C 180,E1 -21194.128,E2 -21194.128} C_VEL
LIN {X 0,Y 211.398,Z 494.085,A -85,B 0,C 180,E1 -21194.796,E2 -21194.796} C_VEL
LIN {X 0,Y 211.091,Z 493.132,A -85,B 0,C 180,E1 -21194.961,E2 -21194.961} C_VEL
LIN {X 0,Y 210.202,Z 488.025,A -85,B 0,C 180,E1 -21199.31,E2 -21199.31} C_VEL
LIN {X 0,Y 209.241,Z 483.274,A -85,B 0,C 180,E1 -21203.713,E2 -21203.713} C_VEL
LIN {X 0,Y 208.26,Z 479.52,A -85,B 0,C 180,E1 -21207.523,E2 -21207.523} C_VEL
LIN {X 0,Y 207.314,Z 475.553,A -85,B 0,C 180,E1 -21211.806,E2 -21211.806} C_VEL
LIN {X 0,Y 206.746,Z 473.347,A -85,B 0,C 180,E1 -21214.585,E2 -21214.585} C_VEL
LIN {X 0,Y 206.777,Z 473.331,A -85,B 0,C 180,E1 -21218.045,E2 -21218.045} C_VEL
LIN {X 0,Y 206.876,Z 473.336,A -85,B 0,C 180,E1 -21222.197,E2 -21222.197} C_VEL
LIN {X 0,Y 206.906,Z 473.336,A -85,B 0,C 180,E1 -21226.245,E2 -21226.245} C_VEL
LIN {X 0,Y 207.123,Z 473.309,A -85,B 0,C 180,E1 -21230.232,E2 -21230.232} C_VEL
LIN {X 0,Y 207.18,Z 473.298,A -85,B 0,C 180,E1 -21232.201,E2 -21232.201} C_VEL
LIN {X 0,Y 207.403,Z 473.268,A -85,B 0,C 180,E1 -21238.058,E2 -21238.058} C_VEL
LIN {X 0,Y 207.51,Z 473.263,A -85,B 0,C 180,E1 -21240,E2 -21240} C_VEL
LIN {X 0,Y 207.373,Z 473.255,A -85,B 0,C 180,E1 -21241.942,E2 -21241.942} C_VEL
LIN {X 0,Y 207.179,Z 473.3,A -85,B 0,C 180,E1 -21247.798,E2 -21247.798} C_VEL
LIN {X 0,Y 206.976,Z 473.299,A -85,B 0,C 180,E1 -21251.755,E2 -21251.755} C_VEL
LIN {X 0,Y 206.864,Z 473.322,A -85,B 0,C 180,E1 -21255.771,E2 -21255.771} C_VEL
LIN {X 0,Y 206.774,Z 473.345,A -85,B 0,C 180,E1 -21259.87,E2 -21259.87} C_VEL
LIN {X 0,Y 206.754,Z 473.356,A -85,B 0,C 180,E1 -21264.073,E2 -21264.073} C_VEL
LIN {X 0,Y 206.736,Z 473.354,A -85,B 0,C 180,E1 -21268.42,E2 -21268.42} C_VEL
LIN {X 0,Y 206.693,Z 473.447,A -85,B 0,C 180,E1 -21272.792,E2 -21272.792} C_VEL
LIN {X 0,Y 208.754,Z 478.962,A -85,B 0,C 180,E1 -21277.3,E2 -21277.3} C_VEL
LIN {X 0,Y 210.451,Z 483.768,A -85,B 0,C 180,E1 -21280.631,E2 -21280.631} C_VEL
LIN {X 0,Y 211.642,Z 488.845,A -85,B 0,C 180,E1 -21283.584,E2 -21283.584} C_VEL
LIN {X 0,Y 212.438,Z 492.74,A -85,B 0,C 180,E1 -21285.599,E2 -21285.599} C_VEL
LIN {X 0,Y 219.742,Z 506.176,A -85,B 0,C 180,E1 -21288.087,E2 -21288.087} C_VEL
LIN {X 0,Y 224.363,Z 516.377,A -85,B 0,C 180,E1 -21289.863,E2 -21289.863} C_VEL
LIN {X 0,Y 226.731,Z 529.116,A -85,B 0,C 180,E1 -21291.577,E2 -21291.577} C_VEL
LIN {X 0,Y 227.636,Z 542.198,A -85,B 0,C 180,E1 -21293.391,E2 -21293.391} C_VEL
LIN {X 0,Y 227.639,Z 555.218,A -85,B 0,C 180,E1 -21295.441,E2 -21295.441} C_VEL
LIN {X 0,Y 227.376,Z 559.629,A -85,B 0,C 180,E1 -21296.198,E2 -21296.198} C_VEL
LIN {X 0,Y 225.978,Z 564.918,A -85,B 0,C 180,E1 -21297.006,E2 -21297.006} C_VEL
LIN {X 0,Y 223.99,Z 569.776,A -85,B 0,C 180,E1 -21297.72,E2 -21297.72} C_VEL
LIN {X 0,Y 219.12,Z 577.386,A -85,B 0,C 180,E1 -21298.774,E2 -21298.774} C_VEL
LIN {X 0,Y 214.147,Z 584.601,A -85,B 0,C 180,E1 -21300,E2 -21300} C_VEL
LIN {X 0,Y 212.036,Z 588.743,A -85,B 0,C 180,E1 -21300.978,E2 -21300.978} C_VEL
LIN {X 0,Y 208.758,Z 597.317,A -85,B 0,C 180,E1 -21303.511,E2 -21303.511} C_VEL
LIN {X 0,Y 205.651,Z 605.036,A -85,B 0,C 180,E1 -21306.328,E2 -21306.328} C_VEL
LIN {X 0,Y 202.771,Z 612.4,A -85,B 0,C 180,E1 -21309.724,E2 -21309.724} C_VEL
LIN {X 0,Y 200.257,Z 618.99,A -85,B 0,C 180,E1 -21313.697,E2 -21313.697} C_VEL
LIN {X 0,Y 198.51,Z 623.927,A -85,B 0,C 180,E1 -21317.738,E2 -21317.738} C_VEL
LIN {X 0,Y 197.571,Z 627.358,A -85,B 0,C 180,E1 -21321.822,E2 -21321.822} C_VEL
LIN {X 0,Y 197.243,Z 629.445,A -85,B 0,C 180,E1 -21326.092,E2 -21326.092} C_VEL
LIN {X 0,Y 197.265,Z 630.051,A -85,B 0,C 180,E1 -21330.003,E2 -21330.003} C_VEL
LIN {X 0,Y 197.249,Z 629.361,A -85,B 0,C 180,E1 -21334.089,E2 -21334.089} C_VEL
LIN {X 0,Y 197.573,Z 627.314,A -85,B 0,C 180,E1 -21338.183,E2 -21338.183} C_VEL
LIN {X 0,Y 198.508,Z 623.866,A -85,B 0,C 180,E1 -21342.267,E2 -21342.267} C_VEL
LIN {X 0,Y 200.261,Z 618.913,A -85,B 0,C 180,E1 -21346.308,E2 -21346.308} C_VEL
LIN {X 0,Y 201.455,Z 615.867,A -85,B 0,C 180,E1 -21348.301,E2 -21348.301} C_VEL
LIN {X 0,Y 204.772,Z 613.814,A -85,B 0,C 180,E1 -21352.183,E2 -21352.183} C_VEL
LIN {X 0,Y 209.323,Z 610.714,A -85,B 0,C 180,E1 -21355.881,E2 -21355.881} C_VEL
LIN {X 0,Y 214.843,Z 606.554,A -85,B 0,C 180,E1 -21359.388,E2 -21359.388} C_VEL
LIN {X 0,Y 221.441,Z 601.293,A -85,B 0,C 180,E1 -21362.655,E2 -21362.655} C_VEL
LIN {X 0,Y 229.092,Z 594.82,A -85,B 0,C 180,E1 -21365.655,E2 -21365.655} C_VEL
LIN {X 0,Y 237.601,Z 587.075,A -85,B 0,C 180,E1 -21368.403,E2 -21368.403} C_VEL
LIN {X 0,Y 245.647,Z 579.139,A -85,B 0,C 180,E1 -21370.61,E2 -21370.61} C_VEL
LIN {X 0,Y 247.886,Z 576.178,A -85,B 0,C 180,E1 -21371.88,E2 -21371.88} C_VEL
LIN {X 0,Y 248.605,Z 574.898,A -85,B 0,C 180,E1 -21372.727,E2 -21372.727} C_VEL
LIN {X 0,Y 248.842,Z 573.243,A -85,B 0,C 180,E1 -21375.084,E2 -21375.084} C_VEL
LIN {X 0,Y 248.654,Z 572.724,A -85,B 0,C 180,E1 -21377.298,E2 -21377.298} C_VEL
LIN {X 0,Y 248.011,Z 573.375,A -85,B 0,C 180,E1 -21379.919,E2 -21379.919} C_VEL
LIN {X 0,Y 247.224,Z 574.463,A -85,B 0,C 180,E1 -21381.288,E2 -21381.288} C_VEL
LIN {X 0,Y 245.559,Z 576.575,A -85,B 0,C 180,E1 -21383.057,E2 -21383.057} C_VEL
LIN {X 0,Y 244.107,Z 578.104,A -85,B 0,C 180,E1 -21383.827,E2 -21383.827} C_VEL
LIN {X 0,Y 235.345,Z 585.543,A -85,B 0,C 180,E1 -21386.464,E2 -21386.464} C_VEL
LIN {X 0,Y 227.384,Z 591.545,A -85,B 0,C 180,E1 -21389.337,E2 -21389.337} C_VEL
LIN {X 0,Y 220.171,Z 596.266,A -85,B 0,C 180,E1 -21392.429,E2 -21392.429} C_VEL
LIN {X 0,Y 215.475,Z 598.926,A -85,B 0,C 180,E1 -21394.912,E2 -21394.912} C_VEL
LIN {X 0,Y 210.051,Z 601.412,A -85,B 0,C 180,E1 -21398.405,E2 -21398.405} C_VEL
LIN {X 0,Y 205.498,Z 602.721,A -85,B 0,C 180,E1 -21402.073,E2 -21402.073} C_VEL
LIN {X 0,Y 202.27,Z 602.769,A -85,B 0,C 180,E1 -21405.923,E2 -21405.923} C_VEL
LIN {X 0,Y 199.761,Z 601.552,A -85,B 0,C 180,E1 -21409.869,E2 -21409.869} C_VEL
LIN {X 0,Y 198.272,Z 598.999,A -85,B 0,C 180,E1 -21413.896,E2 -21413.896} C_VEL
LIN {X 0,Y 197.76,Z 595.101,A -85,B 0,C 180,E1 -21417.964,E2 -21417.964} C_VEL
LIN {X 0,Y 197.641,Z 589.628,A -85,B 0,C 180,E1 -21422.038,E2 -21422.038} C_VEL
LIN {X 0,Y 197.784,Z 583.065,A -85,B 0,C 180,E1 -21425.745,E2 -21425.745} C_VEL
LIN {X 0,Y 198.317,Z 575.451,A -85,B 0,C 180,E1 -21429.176,E2 -21429.176} C_VEL
LIN {X 0,Y 199.181,Z 567.181,A -85,B 0,C 180,E1 -21432.223,E2 -21432.223} C_VEL
LIN {X 0,Y 200.391,Z 557.221,A -85,B 0,C 180,E1 -21435.25,E2 -21435.25} C_VEL
LIN {X 0,Y 202.081,Z 545.187,A -85,B 0,C 180,E1 -21438.241,E2 -21438.241} C_VEL
LIN {X 0,Y 203.782,Z 533.15,A -85,B 0,C 180,E1 -21440.656,E2 -21440.656} C_VEL
LIN {X 0,Y 204.443,Z 528.191,A -85,B 0,C 180,E1 -21441.512,E2 -21441.512} C_VEL
LIN {X 0,Y 202.983,Z 516.779,A -85,B 0,C 180,E1 -21443.329,E2 -21443.329} C_VEL
LIN {X 0,Y 200.968,Z 503.035,A -85,B 0,C 180,E1 -21445.173,E2 -21445.173} C_VEL
LIN {X 0,Y 199.052,Z 488.44,A -85,B 0,C 180,E1 -21446.714,E2 -21446.714} C_VEL
LIN {X 0,Y 198.886,Z 486.452,A -85,B 0,C 180,E1 -21446.92,E2 -21446.92} C_VEL
LIN {X 0,Y 199.501,Z 482.071,A -85,B 0,C 180,E1 -21451.602,E2 -21451.602} C_VEL
LIN {X 0,Y 200.838,Z 483.987,A -85,B 0,C 180,E1 -21454.049,E2 -21454.049} C_VEL
LIN {X 0,Y 202.313,Z 486.49,A -85,B 0,C 180,E1 -21456.964,E2 -21456.964} C_VEL
LIN {X 0,Y 203.212,Z 489.043,A -85,B 0,C 180,E1 -21459.534,E2 -21459.534} C_VEL
LIN {X 0,Y 203.989,Z 493.204,A -85,B 0,C 180,E1 -21463.24,E2 -21463.24} C_VEL
LIN {X 0,Y 205.642,Z 496.646,A -85,B 0,C 180,E1 -21463.901,E2 -21463.901} C_VEL
LIN {X 0,Y 207.153,Z 498.863,A -85,B 0,C 180,E1 -21464.456,E2 -21464.456} C_VEL
LIN {X 0,Y 210.109,Z 504.297,A -85,B 0,C 180,E1 -21465.601,E2 -21465.601} C_VEL
LIN {X 0,Y 212.853,Z 509.926,A -85,B 0,C 180,E1 -21466.744,E2 -21466.744} C_VEL
LIN {X 0,Y 216.522,Z 521.831,A -85,B 0,C 180,E1 -21468.776,E2 -21468.776} C_VEL
LIN {X 0,Y 219.013,Z 533.126,A -85,B 0,C 180,E1 -21470.715,E2 -21470.715} C_VEL
LIN {X 0,Y 220.66,Z 545.936,A -85,B 0,C 180,E1 -21472.995,E2 -21472.995} C_VEL
LIN {X 0,Y 221.157,Z 556.952,A -85,B 0,C 180,E1 -21475.107,E2 -21475.107} C_VEL
LIN {X 0,Y 221.151,Z 560.008,A -85,B 0,C 180,E1 -21475.717,E2 -21475.717} C_VEL
LIN {X 0,Y 217.709,Z 571.687,A -85,B 0,C 180,E1 -21477.813,E2 -21477.813} C_VEL
LIN {X 0,Y 214.167,Z 581.577,A -85,B 0,C 180,E1 -21479.969,E2 -21479.969} C_VEL
LIN {X 0,Y 210.493,Z 591.414,A -85,B 0,C 180,E1 -21482.669,E2 -21482.669} C_VEL
LIN {X 0,Y 207.198,Z 599.577,A -85,B 0,C 180,E1 -21485.446,E2 -21485.446} C_VEL
LIN {X 0,Y 204.22,Z 606.828,A -85,B 0,C 180,E1 -21488.524,E2 -21488.524} C_VEL
LIN {X 0,Y 201.969,Z 612.833,A -85,B 0,C 180,E1 -21491.747,E2 -21491.747} C_VEL
LIN {X 0,Y 199.614,Z 618.546,A -85,B 0,C 180,E1 -21495.73,E2 -21495.73} C_VEL
LIN {X 0,Y 198.199,Z 622.695,A -85,B 0,C 180,E1 -21499.785,E2 -21499.785} C_VEL
LIN {X 0,Y 197.422,Z 625.413,A -85,B 0,C 180,E1 -21503.867,E2 -21503.867} C_VEL
LIN {X 0,Y 197.216,Z 626.774,A -85,B 0,C 180,E1 -21507.955,E2 -21507.955} C_VEL
LIN {X 0,Y 197.249,Z 626.955,A -85,B 0,C 180,E1 -21509.997,E2 -21509.997} C_VEL
LIN {X 0,Y 197.249,Z 626.317,A -85,B 0,C 180,E1 -21514.084,E2 -21514.084} C_VEL
LIN {X 0,Y 197.717,Z 624.333,A -85,B 0,C 180,E1 -21518.172,E2 -21518.172} C_VEL
LIN {X 0,Y 198.8,Z 620.959,A -85,B 0,C 180,E1 -21522.243,E2 -21522.243} C_VEL
LIN {X 0,Y 200.572,Z 616.094,A -85,B 0,C 180,E1 -21526.276,E2 -21526.276} C_VEL
LIN {X 0,Y 202.61,Z 611.378,A -85,B 0,C 180,E1 -21529.237,E2 -21529.237} C_VEL
LIN {X 0,Y 205.242,Z 604.546,A -85,B 0,C 180,E1 -21532.655,E2 -21532.655} C_VEL
LIN {X 0,Y 208.723,Z 596.059,A -85,B 0,C 180,E1 -21535.956,E2 -21535.956} C_VEL
LIN {X 0,Y 212.184,Z 587.18,A -85,B 0,C 180,E1 -21538.7,E2 -21538.7} C_VEL
LIN {X 0,Y 216.161,Z 576.426,A -85,B 0,C 180,E1 -21541.343,E2 -21541.343} C_VEL
LIN {X 0,Y 219.809,Z 565.368,A -85,B 0,C 180,E1 -21543.501,E2 -21543.501} C_VEL
LIN {X 0,Y 221.234,Z 559.475,A -85,B 0,C 180,E1 -21544.527,E2 -21544.527} C_VEL
LIN {X 0,Y 220.892,Z 548.05,A -85,B 0,C 180,E1 -21546.761,E2 -21546.761} C_VEL
LIN {X 0,Y 219.735,Z 537.274,A -85,B 0,C 180,E1 -21548.709,E2 -21548.709} C_VEL
LIN {X 0,Y 217.982,Z 527.887,A -85,B 0,C 180,E1 -21550.345,E2 -21550.345} C_VEL
LIN {X 0,Y 214.795,Z 515.635,A -85,B 0,C 180,E1 -21552.429,E2 -21552.429} C_VEL
LIN {X 0,Y 212.019,Z 508.031,A -85,B 0,C 180,E1 -21553.78,E2 -21553.78} C_VEL
LIN {X 0,Y 208.883,Z 501.974,A -85,B 0,C 180,E1 -21555.044,E2 -21555.044} C_VEL
LIN {X 0,Y 206.537,Z 497.704,A -85,B 0,C 180,E1 -21555.963,E2 -21555.963} C_VEL
LIN {X 0,Y 204.402,Z 494.271,A -85,B 0,C 180,E1 -21556.762,E2 -21556.762} C_VEL
LIN {X 0,Y 203.996,Z 493.083,A -85,B 0,C 180,E1 -21557.006,E2 -21557.006} C_VEL
LIN {X 0,Y 203.113,Z 488.197,A -85,B 0,C 180,E1 -21561.477,E2 -21561.477} C_VEL
LIN {X 0,Y 202.298,Z 484.6,A -85,B 0,C 180,E1 -21565.024,E2 -21565.024} C_VEL
LIN {X 0,Y 201.477,Z 481.414,A -85,B 0,C 180,E1 -21568.45,E2 -21568.45} C_VEL
LIN {X 0,Y 200.544,Z 477.566,A -85,B 0,C 180,E1 -21572.898,E2 -21572.898} C_VEL
LIN {X 0,Y 199.72,Z 474.211,A -85,B 0,C 180,E1 -21577.5,E2 -21577.5} C_VEL
LIN {X 0,Y 199.829,Z 474.214,A -85,B 0,C 180,E1 -21581.72,E2 -21581.72} C_VEL
LIN {X 0,Y 199.842,Z 474.213,A -85,B 0,C 180,E1 -21585.749,E2 -21585.749} C_VEL
LIN {X 0,Y 200.066,Z 474.19,A -85,B 0,C 180,E1 -21589.884,E2 -21589.884} C_VEL
LIN {X 0,Y 200.034,Z 474.189,A -85,B 0,C 180,E1 -21593.949,E2 -21593.949} C_VEL
LIN {X 0,Y 200.339,Z 474.148,A -85,B 0,C 180,E1 -21597.989,E2 -21597.989} C_VEL
LIN {X 0,Y 200.474,Z 474.14,A -85,B 0,C 180,E1 -21600,E2 -21600} C_VEL
LIN {X 0,Y 200.022,Z 474.159,A -85,B 0,C 180,E1 -21604.029,E2 -21604.029} C_VEL
LIN {X 0,Y 200.122,Z 474.173,A -85,B 0,C 180,E1 -21608.075,E2 -21608.075} C_VEL
LIN {X 0,Y 199.908,Z 474.182,A -85,B 0,C 180,E1 -21612.177,E2 -21612.177} C_VEL
LIN {X 0,Y 199.799,Z 474.195,A -85,B 0,C 180,E1 -21616.344,E2 -21616.344} C_VEL
LIN {X 0,Y 199.691,Z 474.237,A -85,B 0,C 180,E1 -21620.606,E2 -21620.606} C_VEL
LIN {X 0,Y 199.664,Z 474.234,A -85,B 0,C 180,E1 -21624.985,E2 -21624.985} C_VEL
LIN {X 0,Y 199.668,Z 474.263,A -85,B 0,C 180,E1 -21629.668,E2 -21629.668} C_VEL
LIN {X 0,Y 201.763,Z 480.135,A -85,B 0,C 180,E1 -21635.082,E2 -21635.082} C_VEL
LIN {X 0,Y 203.306,Z 484.467,A -85,B 0,C 180,E1 -21638.479,E2 -21638.479} C_VEL
LIN {X 0,Y 204.488,Z 487.912,A -85,B 0,C 180,E1 -21640.882,E2 -21640.882} C_VEL
LIN {X 0,Y 205.574,Z 492.779,A -85,B 0,C 180,E1 -21643.69,E2 -21643.69} C_VEL
LIN {X 0,Y 213.385,Z 506.983,A -85,B 0,C 180,E1 -21646.584,E2 -21646.584} C_VEL
LIN {X 0,Y 218.896,Z 519.288,A -85,B 0,C 180,E1 -21648.894,E2 -21648.894} C_VEL
LIN {X 0,Y 220.609,Z 528.301,A -85,B 0,C 180,E1 -21650.211,E2 -21650.211} C_VEL
LIN {X 0,Y 221.586,Z 539.157,A -85,B 0,C 180,E1 -21651.778,E2 -21651.778} C_VEL
LIN {X 0,Y 221.629,Z 552.435,A -85,B 0,C 180,E1 -21653.872,E2 -21653.872} C_VEL
LIN {X 0,Y 221.094,Z 561.146,A -85,B 0,C 180,E1 -21655.406,E2 -21655.406} C_VEL
LIN {X 0,Y 217.826,Z 572.262,A -85,B 0,C 180,E1 -21657.29,E2 -21657.29} C_VEL
LIN {X 0,Y 214.356,Z 582.608,A -85,B 0,C 180,E1 -21659.46,E2 -21659.46} C_VEL
LIN {X 0,Y 212.036,Z 588.743,A -85,B 0,C 180,E1 -21660.978,E2 -21660.978} C_VEL
LIN {X 0,Y 209.923,Z 592.794,A -85,B 0,C 180,E1 -21662.022,E2 -21662.022} C_VEL
LIN {X 0,Y 204.866,Z 598.973,A -85,B 0,C 180,E1 -21663.651,E2 -21663.651} C_VEL
LIN {X 0,Y 199.877,Z 604.68,A -85,B 0,C 180,E1 -21665.459,E2 -21665.459} C_VEL
LIN {X 0,Y 197.911,Z 607.837,A -85,B 0,C 180,E1 -21666.763,E2 -21666.763} C_VEL
LIN {X 0,Y 195.343,Z 614.15,A -85,B 0,C 180,E1 -21670.017,E2 -21670.017} C_VEL
LIN {X 0,Y 193.416,Z 618.936,A -85,B 0,C 180,E1 -21673.104,E2 -21673.104} C_VEL
LIN {X 0,Y 191.55,Z 623.873,A -85,B 0,C 180,E1 -21677.286,E2 -21677.286} C_VEL
LIN {X 0,Y 190.517,Z 627.303,A -85,B 0,C 180,E1 -21681.517,E2 -21681.517} C_VEL
LIN {X 0,Y 190.161,Z 629.329,A -85,B 0,C 180,E1 -21685.764,E2 -21685.764} C_VEL
LIN {X 0,Y 190.173,Z 629.996,A -85,B 0,C 180,E1 -21690.003,E2 -21690.003} C_VEL
LIN {X 0,Y 190.163,Z 629.305,A -85,B 0,C 180,E1 -21694.242,E2 -21694.242} C_VEL
LIN {X 0,Y 190.52,Z 627.258,A -85,B 0,C 180,E1 -21698.488,E2 -21698.488} C_VEL
LIN {X 0,Y 191.548,Z 623.81,A -85,B 0,C 180,E1 -21702.72,E2 -21702.72} C_VEL
LIN {X 0,Y 193.426,Z 618.857,A -85,B 0,C 180,E1 -21706.901,E2 -21706.901} C_VEL
LIN {X 0,Y 194.883,Z 615.604,A -85,B 0,C 180,E1 -21709.215,E2 -21709.215} C_VEL
LIN {X 0,Y 198.193,Z 613.967,A -85,B 0,C 180,E1 -21712.961,E2 -21712.961} C_VEL
LIN {X 0,Y 202.977,Z 611.213,A -85,B 0,C 180,E1 -21716.754,E2 -21716.754} C_VEL
LIN {X 0,Y 210.412,Z 606.297,A -85,B 0,C 180,E1 -21721.182,E2 -21721.182} C_VEL
LIN {X 0,Y 217.499,Z 601.185,A -85,B 0,C 180,E1 -21724.438,E2 -21724.438} C_VEL
LIN {X 0,Y 225.622,Z 594.912,A -85,B 0,C 180,E1 -21727.405,E2 -21727.405} C_VEL
LIN {X 0,Y 235.79,Z 586.352,A -85,B 0,C 180,E1 -21730.415,E2 -21730.415} C_VEL
LIN {X 0,Y 240.621,Z 582.007,A -85,B 0,C 180,E1 -21731.645,E2 -21731.645} C_VEL
LIN {X 0,Y 241.549,Z 581.05,A -85,B 0,C 180,E1 -21732.008,E2 -21732.008} C_VEL
LIN {X 0,Y 242.905,Z 579.375,A -85,B 0,C 180,E1 -21732.915,E2 -21732.915} C_VEL
LIN {X 0,Y 243.145,Z 578.548,A -85,B 0,C 180,E1 -21733.927,E2 -21733.927} C_VEL
LIN {X 0,Y 243.229,Z 577.496,A -85,B 0,C 180,E1 -21736.253,E2 -21736.253} C_VEL
LIN {X 0,Y 242.761,Z 577.54,A -85,B 0,C 180,E1 -21738.828,E2 -21738.828} C_VEL
LIN {X 0,Y 242.106,Z 578.234,A -85,B 0,C 180,E1 -21740.31,E2 -21740.31} C_VEL
LIN {X 0,Y 240.432,Z 579.938,A -85,B 0,C 180,E1 -21742.132,E2 -21742.132} C_VEL
LIN {X 0,Y 238.835,Z 581.422,A -85,B 0,C 180,E1 -21742.898,E2 -21742.898} C_VEL
LIN {X 0,Y 229.793,Z 588.23,A -85,B 0,C 180,E1 -21745.542,E2 -21745.542} C_VEL
LIN {X 0,Y 221.545,Z 593.743,A -85,B 0,C 180,E1 -21748.438,E2 -21748.438} C_VEL
LIN {X 0,Y 215.867,Z 597.068,A -85,B 0,C 180,E1 -21750.767,E2 -21750.767} C_VEL
LIN {X 0,Y 209.193,Z 600.342,A -85,B 0,C 180,E1 -21754.104,E2 -21754.104} C_VEL
LIN {X 0,Y 203.555,Z 602.451,A -85,B 0,C 180,E1 -21757.68,E2 -21757.68} C_VEL
LIN {X 0,Y 198.809,Z 603.381,A -85,B 0,C 180,E1 -21761.449,E2 -21761.449} C_VEL
LIN {X 0,Y 195.408,Z 603.079,A -85,B 0,C 180,E1 -21765.418,E2 -21765.418} C_VEL
LIN {X 0,Y 192.795,Z 601.546,A -85,B 0,C 180,E1 -21769.498,E2 -21769.498} C_VEL
LIN {X 0,Y 191.222,Z 598.732,A -85,B 0,C 180,E1 -21773.67,E2 -21773.67} C_VEL
LIN {X 0,Y 190.7,Z 594.528,A -85,B 0,C 180,E1 -21777.888,E2 -21777.888} C_VEL
LIN {X 0,Y 190.561,Z 590.37,A -85,B 0,C 180,E1 -21781.057,E2 -21781.057} C_VEL
LIN {X 0,Y 190.634,Z 584.076,A -85,B 0,C 180,E1 -21784.821,E2 -21784.821} C_VEL
LIN {X 0,Y 191.114,Z 576.462,A -85,B 0,C 180,E1 -21788.459,E2 -21788.459} C_VEL
LIN {X 0,Y 192.082,Z 566.969,A -85,B 0,C 180,E1 -21792.145,E2 -21792.145} C_VEL
LIN {X 0,Y 193.304,Z 556.865,A -85,B 0,C 180,E1 -21795.283,E2 -21795.283} C_VEL
LIN {X 0,Y 195.023,Z 544.708,A -85,B 0,C 180,E1 -21798.38,E2 -21798.38} C_VEL
LIN {X 0,Y 196.783,Z 532.309,A -85,B 0,C 180,E1 -21800.925,E2 -21800.925} C_VEL
LIN {X 0,Y 197.33,Z 527.648,A -85,B 0,C 180,E1 -21801.758,E2 -21801.758} C_VEL
LIN {X 0,Y 195.404,Z 513.638,A -85,B 0,C 180,E1 -21804.012,E2 -21804.012} C_VEL
LIN {X 0,Y 193.264,Z 498.854,A -85,B 0,C 180,E1 -21805.937,E2 -21805.937} C_VEL
LIN {X 0,Y 191.859,Z 486.646,A -85,B 0,C 180,E1 -21807.251,E2 -21807.251} C_VEL
LIN {X 0,Y 192.248,Z 483.942,A -85,B 0,C 180,E1 -21810.251,E2 -21810.251} C_VEL
LIN {X 0,Y 194.006,Z 486.359,A -85,B 0,C 180,E1 -21813.568,E2 -21813.568} C_VEL
LIN {X 0,Y 195.48,Z 488.622,A -85,B 0,C 180,E1 -21816.386,E2 -21816.386} C_VEL
LIN {X 0,Y 196.401,Z 490.828,A -85,B 0,C 180,E1 -21818.771,E2 -21818.771} C_VEL
LIN {X 0,Y 196.956,Z 493.396,A -85,B 0,C 180,E1 -21821.032,E2 -21821.032} C_VEL
LIN {X 0,Y 198.773,Z 496.827,A -85,B 0,C 180,E1 -21821.816,E2 -21821.816} C_VEL
LIN {X 0,Y 200.343,Z 499.077,A -85,B 0,C 180,E1 -21822.451,E2 -21822.451} C_VEL
LIN {X 0,Y 205.592,Z 508.688,A -85,B 0,C 180,E1 -21824.708,E2 -21824.708} C_VEL
LIN {X 0,Y 208.153,Z 514.46,A -85,B 0,C 180,E1 -21825.934,E2 -21825.934} C_VEL
LIN {X 0,Y 211.158,Z 524.98,A -85,B 0,C 180,E1 -21827.852,E2 -21827.852} C_VEL
LIN {X 0,Y 213.471,Z 536.565,A -85,B 0,C 180,E1 -21829.973,E2 -21829.973} C_VEL
LIN {X 0,Y 214.693,Z 548.089,A -85,B 0,C 180,E1 -21832.15,E2 -21832.15} C_VEL
LIN {X 0,Y 214.985,Z 559.15,A -85,B 0,C 180,E1 -21834.397,E2 -21834.397} C_VEL
LIN {X 0,Y 214.729,Z 562.276,A -85,B 0,C 180,E1 -21835.042,E2 -21835.042} C_VEL
LIN {X 0,Y 210.948,Z 573.84,A -85,B 0,C 180,E1 -21837.219,E2 -21837.219} C_VEL
LIN {X 0,Y 207.308,Z 583.384,A -85,B 0,C 180,E1 -21839.432,E2 -21839.432} C_VEL
LIN {X 0,Y 203.589,Z 592.933,A -85,B 0,C 180,E1 -21842.221,E2 -21842.221} C_VEL
LIN {X 0,Y 200.193,Z 600.847,A -85,B 0,C 180,E1 -21845.083,E2 -21845.083} C_VEL
LIN {X 0,Y 197.422,Z 607.296,A -85,B 0,C 180,E1 -21847.975,E2 -21847.975} C_VEL
LIN {X 0,Y 195.22,Z 612.889,A -85,B 0,C 180,E1 -21851.092,E2 -21851.092} C_VEL
LIN {X 0,Y 192.698,Z 618.603,A -85,B 0,C 180,E1 -21855.206,E2 -21855.206} C_VEL
LIN {X 0,Y 191.206,Z 622.752,A -85,B 0,C 180,E1 -21859.407,E2 -21859.407} C_VEL
LIN {X 0,Y 190.363,Z 625.469,A -85,B 0,C 180,E1 -21863.638,E2 -21863.638} C_VEL
LIN {X 0,Y 190.129,Z 626.83,A -85,B 0,C 180,E1 -21867.879,E2 -21867.879} C_VEL
LIN {X 0,Y 190.158,Z 627.01,A -85,B 0,C 180,E1 -21869.997,E2 -21869.997} C_VEL
LIN {X 0,Y 190.165,Z 626.373,A -85,B 0,C 180,E1 -21874.236,E2 -21874.236} C_VEL
LIN {X 0,Y 190.689,Z 624.388,A -85,B 0,C 180,E1 -21878.475,E2 -21878.475} C_VEL
LIN {X 0,Y 191.82,Z 621.014,A -85,B 0,C 180,E1 -21882.696,E2 -21882.696} C_VEL
LIN {X 0,Y 193.761,Z 616.147,A -85,B 0,C 180,E1 -21886.865,E2 -21886.865} C_VEL
LIN {X 0,Y 195.871,Z 611.431,A -85,B 0,C 180,E1 -21889.927,E2 -21889.927} C_VEL
LIN {X 0,Y 198.684,Z 604.597,A -85,B 0,C 180,E1 -21893.447,E2 -21893.447} C_VEL
LIN {X 0,Y 202.351,Z 596.108,A -85,B 0,C 180,E1 -21896.838,E2 -21896.838} C_VEL
LIN {X 0,Y 205.952,Z 587.228,A -85,B 0,C 180,E1 -21899.654,E2 -21899.654} C_VEL
LIN {X 0,Y 210.128,Z 576.47,A -85,B 0,C 180,E1 -21902.35,E2 -21902.35} C_VEL
LIN {X 0,Y 214.184,Z 564.483,A -85,B 0,C 180,E1 -21904.713,E2 -21904.713} C_VEL
LIN {X 0,Y 215,Z 561.018,A -85,B 0,C 180,E1 -21905.345,E2 -21905.345} C_VEL
LIN {X 0,Y 214.828,Z 549.249,A -85,B 0,C 180,E1 -21907.762,E2 -21907.762} C_VEL
LIN {X 0,Y 213.661,Z 537.676,A -85,B 0,C 180,E1 -21909.967,E2 -21909.967} C_VEL
LIN {X 0,Y 211.402,Z 525.956,A -85,B 0,C 180,E1 -21912.126,E2 -21912.126} C_VEL
LIN {X 0,Y 208.089,Z 514.012,A -85,B 0,C 180,E1 -21914.297,E2 -21914.297} C_VEL
LIN {X 0,Y 204.557,Z 506.65,A -85,B 0,C 180,E1 -21915.928,E2 -21915.928} C_VEL
LIN {X 0,Y 202.111,Z 502.167,A -85,B 0,C 180,E1 -21916.983,E2 -21916.983} C_VEL
LIN {X 0,Y 199.487,Z 497.67,A -85,B 0,C 180,E1 -21918.094,E2 -21918.094} C_VEL
LIN {X 0,Y 197.314,Z 494.205,A -85,B 0,C 180,E1 -21918.994,E2 -21918.994} C_VEL
LIN {X 0,Y 196.929,Z 493.167,A -85,B 0,C 180,E1 -21919.181,E2 -21919.181} C_VEL
LIN {X 0,Y 196.058,Z 488.539,A -85,B 0,C 180,E1 -21923.739,E2 -21923.739} C_VEL
LIN {X 0,Y 195.213,Z 485.184,A -85,B 0,C 180,E1 -21927.314,E2 -21927.314} C_VEL
LIN {X 0,Y 194.27,Z 481.326,A -85,B 0,C 180,E1 -21931.946,E2 -21931.946} C_VEL
LIN {X 0,Y 193.418,Z 477.852,A -85,B 0,C 180,E1 -21936.441,E2 -21936.441} C_VEL
LIN {X 0,Y 192.717,Z 475.106,A -85,B 0,C 180,E1 -21940.839,E2 -21940.839} C_VEL
LIN {X 0,Y 192.768,Z 475.092,A -85,B 0,C 180,E1 -21945.214,E2 -21945.214} C_VEL
LIN {X 0,Y 193.011,Z 475.067,A -85,B 0,C 180,E1 -21949.51,E2 -21949.51} C_VEL
LIN {X 0,Y 192.997,Z 475.067,A -85,B 0,C 180,E1 -21953.728,E2 -21953.728} C_VEL
LIN {X 0,Y 193.278,Z 475.027,A -85,B 0,C 180,E1 -21957.916,E2 -21957.916} C_VEL
LIN {X 0,Y 193.437,Z 475.016,A -85,B 0,C 180,E1 -21960,E2 -21960} C_VEL
LIN {X 0,Y 192.969,Z 475.038,A -85,B 0,C 180,E1 -21964.177,E2 -21964.177} C_VEL
LIN {X 0,Y 193.069,Z 475.045,A -85,B 0,C 180,E1 -21968.372,E2 -21968.372} C_VEL
LIN {X 0,Y 192.847,Z 475.067,A -85,B 0,C 180,E1 -21972.63,E2 -21972.63} C_VEL
LIN {X 0,Y 192.751,Z 475.069,A -85,B 0,C 180,E1 -21976.959,E2 -21976.959} C_VEL
LIN {X 0,Y 192.627,Z 475.112,A -85,B 0,C 180,E1 -21981.398,E2 -21981.398} C_VEL
LIN {X 0,Y 192.655,Z 475.111,A -85,B 0,C 180,E1 -21984.226,E2 -21984.226} C_VEL
LIN {X 0,Y 192.632,Z 475.336,A -85,B 0,C 180,E1 -21986.255,E2 -21986.255} C_VEL
LIN {X 0,Y 193.703,Z 478.063,A -85,B 0,C 180,E1 -21989.457,E2 -21989.457} C_VEL
LIN {X 0,Y 195.335,Z 482.938,A -85,B 0,C 180,E1 -21994.16,E2 -21994.16} C_VEL
LIN {X 0,Y 197.26,Z 488.153,A -85,B 0,C 180,E1 -21998.393,E2 -21998.393} C_VEL
LIN {X 0,Y 198.619,Z 492.665,A -85,B 0,C 180,E1 -22001.534,E2 -22001.534} C_VEL
LIN {X 0,Y 201.204,Z 497.137,A -85,B 0,C 180,E1 -22002.592,E2 -22002.592} C_VEL
LIN {X 0,Y 207.054,Z 507.865,A -85,B 0,C 180,E1 -22004.969,E2 -22004.969} C_VEL
LIN {X 0,Y 211.998,Z 518.54,A -85,B 0,C 180,E1 -22007.178,E2 -22007.178} C_VEL
LIN {X 0,Y 214.113,Z 524.464,A -85,B 0,C 180,E1 -22008.309,E2 -22008.309} C_VEL
LIN {X 0,Y 215.543,Z 536.094,A -85,B 0,C 180,E1 -22010.08,E2 -22010.08} C_VEL
LIN {X 0,Y 215.77,Z 548.587,A -85,B 0,C 180,E1 -22012.058,E2 -22012.058} C_VEL
LIN {X 0,Y 215.121,Z 560.968,A -85,B 0,C 180,E1 -22014.273,E2 -22014.273} C_VEL
LIN {X 0,Y 213.352,Z 567.518,A -85,B 0,C 180,E1 -22015.378,E2 -22015.378} C_VEL
LIN {X 0,Y 209.66,Z 578.68,A -85,B 0,C 180,E1 -22017.569,E2 -22017.569} C_VEL
LIN {X 0,Y 205.48,Z 589.609,A -85,B 0,C 180,E1 -22020.271,E2 -22020.271} C_VEL
LIN {X 0,Y 201.812,Z 598.619,A -85,B 0,C 180,E1 -22023.085,E2 -22023.085} C_VEL
LIN {X 0,Y 198.169,Z 607.222,A -85,B 0,C 180,E1 -22026.489,E2 -22026.489} C_VEL
LIN {X 0,Y 197.911,Z 607.837,A -85,B 0,C 180,E1 -22026.763,E2 -22026.763} C_VEL
LIN {X 0,Y 196.036,Z 610.871,A -85,B 0,C 180,E1 -22028.136,E2 -22028.136} C_VEL
LIN {X 0,Y 191.462,Z 615.371,A -85,B 0,C 180,E1 -22030.375,E2 -22030.375} C_VEL
LIN {X 0,Y 187.062,Z 619.271,A -85,B 0,C 180,E1 -22032.803,E2 -22032.803} C_VEL
LIN {X 0,Y 185.506,Z 621.344,A -85,B 0,C 180,E1 -22034.442,E2 -22034.442} C_VEL
LIN {X 0,Y 183.927,Z 625.714,A -85,B 0,C 180,E1 -22038.989,E2 -22038.989} C_VEL
LIN {X 0,Y 183.207,Z 628.432,A -85,B 0,C 180,E1 -22043.394,E2 -22043.394} C_VEL
LIN {X 0,Y 183.04,Z 629.776,A -85,B 0,C 180,E1 -22047.802,E2 -22047.802} C_VEL
LIN {X 0,Y 183.084,Z 629.94,A -85,B 0,C 180,E1 -22050.003,E2 -22050.003} C_VEL
LIN {X 0,Y 183.077,Z 629.249,A -85,B 0,C 180,E1 -22054.406,E2 -22054.406} C_VEL
LIN {X 0,Y 183.488,Z 627.202,A -85,B 0,C 180,E1 -22058.816,E2 -22058.816} C_VEL
LIN {X 0,Y 184.585,Z 623.754,A -85,B 0,C 180,E1 -22063.208,E2 -22063.208} C_VEL
LIN {X 0,Y 186.611,Z 618.801,A -85,B 0,C 180,E1 -22067.538,E2 -22067.538} C_VEL
LIN {X 0,Y 188.169,Z 615.372,A -85,B 0,C 180,E1 -22069.929,E2 -22069.929} C_VEL
LIN {X 0,Y 191.664,Z 613.998,A -85,B 0,C 180,E1 -22073.791,E2 -22073.791} C_VEL
LIN {X 0,Y 196.664,Z 611.59,A -85,B 0,C 180,E1 -22077.685,E2 -22077.685} C_VEL
LIN {X 0,Y 204.418,Z 607.179,A -85,B 0,C 180,E1 -22082.204,E2 -22082.204} C_VEL
LIN {X 0,Y 211.775,Z 602.497,A -85,B 0,C 180,E1 -22085.506,E2 -22085.506} C_VEL
LIN {X 0,Y 220.177,Z 596.712,A -85,B 0,C 180,E1 -22088.497,E2 -22088.497} C_VEL
LIN {X 0,Y 229.437,Z 589.758,A -85,B 0,C 180,E1 -22091.194,E2 -22091.194} C_VEL
LIN {X 0,Y 234.38,Z 585.818,A -85,B 0,C 180,E1 -22092.431,E2 -22092.431} C_VEL
LIN {X 0,Y 236.664,Z 583.877,A -85,B 0,C 180,E1 -22093.082,E2 -22093.082} C_VEL
LIN {X 0,Y 237.439,Z 582.414,A -85,B 0,C 180,E1 -22094.734,E2 -22094.734} C_VEL
LIN {X 0,Y 237.389,Z 581.704,A -85,B 0,C 180,E1 -22097.084,E2 -22097.084} C_VEL
LIN {X 0,Y 236.817,Z 582,A -85,B 0,C 180,E1 -22099.24,E2 -22099.24} C_VEL
LIN {X 0,Y 235.268,Z 583.315,A -85,B 0,C 180,E1 -22101.148,E2 -22101.148} C_VEL
LIN {X 0,Y 234.392,Z 584.017,A -85,B 0,C 180,E1 -22101.672,E2 -22101.672} C_VEL
LIN {X 0,Y 224.065,Z 591.039,A -85,B 0,C 180,E1 -22104.641,E2 -22104.641} C_VEL
LIN {X 0,Y 213.74,Z 596.934,A -85,B 0,C 180,E1 -22108.258,E2 -22108.258} C_VEL
LIN {X 0,Y 206.294,Z 600.409,A -85,B 0,C 180,E1 -22111.514,E2 -22111.514} C_VEL
LIN {X 0,Y 199.889,Z 602.698,A -85,B 0,C 180,E1 -22115.045,E2 -22115.045} C_VEL
LIN {X 0,Y 194.482,Z 603.855,A -85,B 0,C 180,E1 -22118.816,E2 -22118.816} C_VEL
LIN {X 0,Y 190.227,Z 603.821,A -85,B 0,C 180,E1 -22122.809,E2 -22122.809} C_VEL
LIN {X 0,Y 187.031,Z 602.574,A -85,B 0,C 180,E1 -22126.97,E2 -22126.97} C_VEL
LIN {X 0,Y 184.827,Z 600.065,A -85,B 0,C 180,E1 -22131.252,E2 -22131.252} C_VEL
LIN {X 0,Y 183.826,Z 596.274,A -85,B 0,C 180,E1 -22135.615,E2 -22135.615} C_VEL
LIN {X 0,Y 183.548,Z 592.467,A -85,B 0,C 180,E1 -22138.903,E2 -22138.903} C_VEL
LIN {X 0,Y 183.526,Z 587.752,A -85,B 0,C 180,E1 -22142.195,E2 -22142.195} C_VEL
LIN {X 0,Y 183.702,Z 581.197,A -85,B 0,C 180,E1 -22145.882,E2 -22145.882} C_VEL
LIN {X 0,Y 184.263,Z 573.626,A -85,B 0,C 180,E1 -22149.329,E2 -22149.329} C_VEL
LIN {X 0,Y 185.158,Z 564.951,A -85,B 0,C 180,E1 -22152.607,E2 -22152.607} C_VEL
LIN {X 0,Y 186.522,Z 554.609,A -85,B 0,C 180,E1 -22155.853,E2 -22155.853} C_VEL
LIN {X 0,Y 188.171,Z 543.036,A -85,B 0,C 180,E1 -22158.792,E2 -22158.792} C_VEL
LIN {X 0,Y 189.961,Z 530.29,A -85,B 0,C 180,E1 -22161.429,E2 -22161.429} C_VEL
LIN {X 0,Y 190.127,Z 527.138,A -85,B 0,C 180,E1 -22161.995,E2 -22161.995} C_VEL
LIN {X 0,Y 188.217,Z 513.54,A -85,B 0,C 180,E1 -22164.251,E2 -22164.251} C_VEL
LIN {X 0,Y 186.087,Z 498.577,A -85,B 0,C 180,E1 -22166.274,E2 -22166.274} C_VEL
LIN {X 0,Y 184.815,Z 486.785,A -85,B 0,C 180,E1 -22167.596,E2 -22167.596} C_VEL
LIN {X 0,Y 184.948,Z 485.892,A -85,B 0,C 180,E1 -22168.759,E2 -22168.759} C_VEL
LIN {X 0,Y 187.754,Z 489.593,A -85,B 0,C 180,E1 -22174.159,E2 -22174.159} C_VEL
LIN {X 0,Y 188.979,Z 491.425,A -85,B 0,C 180,E1 -22176.515,E2 -22176.515} C_VEL
LIN {X 0,Y 189.751,Z 493.281,A -85,B 0,C 180,E1 -22178.463,E2 -22178.463} C_VEL
LIN {X 0,Y 191.774,Z 496.917,A -85,B 0,C 180,E1 -22179.431,E2 -22179.431} C_VEL
LIN {X 0,Y 193.393,Z 498.994,A -85,B 0,C 180,E1 -22180.145,E2 -22180.145} C_VEL
LIN {X 0,Y 195.901,Z 503.221,A -85,B 0,C 180,E1 -22181.302,E2 -22181.302} C_VEL
LIN {X 0,Y 201.176,Z 513.444,A -85,B 0,C 180,E1 -22183.871,E2 -22183.871} C_VEL
LIN {X 0,Y 203.423,Z 518.828,A -85,B 0,C 180,E1 -22185.093,E2 -22185.093} C_VEL
LIN {X 0,Y 206.079,Z 529.472,A -85,B 0,C 180,E1 -22187.156,E2 -22187.156} C_VEL
LIN {X 0,Y 207.968,Z 540.831,A -85,B 0,C 180,E1 -22189.388,E2 -22189.388} C_VEL
LIN {X 0,Y 208.819,Z 552.591,A -85,B 0,C 180,E1 -22191.771,E2 -22191.771} C_VEL
LIN {X 0,Y 208.755,Z 562.379,A -85,B 0,C 180,E1 -22193.9,E2 -22193.9} C_VEL
LIN {X 0,Y 206.964,Z 568.421,A -85,B 0,C 180,E1 -22195.035,E2 -22195.035} C_VEL
LIN {X 0,Y 202.7,Z 579.832,A -85,B 0,C 180,E1 -22197.49,E2 -22197.49} C_VEL
LIN {X 0,Y 198.564,Z 590.041,A -85,B 0,C 180,E1 -22200.293,E2 -22200.293} C_VEL
LIN {X 0,Y 194.906,Z 598.459,A -85,B 0,C 180,E1 -22203.207,E2 -22203.207} C_VEL
LIN {X 0,Y 191.652,Z 605.447,A -85,B 0,C 180,E1 -22206.208,E2 -22206.208} C_VEL
LIN {X 0,Y 189.219,Z 611.238,A -85,B 0,C 180,E1 -22209.336,E2 -22209.336} C_VEL
LIN {X 0,Y 186.393,Z 617.414,A -85,B 0,C 180,E1 -22213.571,E2 -22213.571} C_VEL
LIN {X 0,Y 184.9,Z 620.919,A -85,B 0,C 180,E1 -22216.814,E2 -22216.814} C_VEL
LIN {X 0,Y 183.661,Z 624.339,A -85,B 0,C 180,E1 -22221.193,E2 -22221.193} C_VEL
LIN {X 0,Y 183.082,Z 626.372,A -85,B 0,C 180,E1 -22225.594,E2 -22225.594} C_VEL
LIN {X 0,Y 183.069,Z 627.066,A -85,B 0,C 180,E1 -22229.997,E2 -22229.997} C_VEL
LIN {X 0,Y 183.081,Z 626.428,A -85,B 0,C 180,E1 -22234.4,E2 -22234.4} C_VEL
LIN {X 0,Y 183.657,Z 624.443,A -85,B 0,C 180,E1 -22238.802,E2 -22238.802} C_VEL
LIN {X 0,Y 184.864,Z 621.068,A -85,B 0,C 180,E1 -22243.182,E2 -22243.182} C_VEL
LIN {X 0,Y 186.969,Z 616.201,A -85,B 0,C 180,E1 -22247.497,E2 -22247.497} C_VEL
LIN {X 0,Y 189.153,Z 611.484,A -85,B 0,C 180,E1 -22250.666,E2 -22250.666} C_VEL
LIN {X 0,Y 192.152,Z 604.649,A -85,B 0,C 180,E1 -22254.294,E2 -22254.294} C_VEL
LIN {X 0,Y 196.025,Z 596.158,A -85,B 0,C 180,E1 -22257.777,E2 -22257.777} C_VEL
LIN {X 0,Y 199.795,Z 587.276,A -85,B 0,C 180,E1 -22260.664,E2 -22260.664} C_VEL
LIN {X 0,Y 204.157,Z 576.514,A -85,B 0,C 180,E1 -22263.418,E2 -22263.418} C_VEL
LIN {X 0,Y 208.366,Z 564.523,A -85,B 0,C 180,E1 -22265.829,E2 -22265.829} C_VEL
LIN {X 0,Y 208.818,Z 562.2,A -85,B 0,C 180,E1 -22266.286,E2 -22266.286} C_VEL
LIN {X 0,Y 208.874,Z 551.703,A -85,B 0,C 180,E1 -22268.554,E2 -22268.554} C_VEL
LIN {X 0,Y 208.051,Z 541.008,A -85,B 0,C 180,E1 -22270.726,E2 -22270.726} C_VEL
LIN {X 0,Y 206.16,Z 529.546,A -85,B 0,C 180,E1 -22272.98,E2 -22272.98} C_VEL
LIN {X 0,Y 203.169,Z 517.827,A -85,B 0,C 180,E1 -22275.273,E2 -22275.273} C_VEL
LIN {X 0,Y 199.721,Z 510.341,A -85,B 0,C 180,E1 -22277.06,E2 -22277.06} C_VEL
LIN {X 0,Y 195.599,Z 502.768,A -85,B 0,C 180,E1 -22279.021,E2 -22279.021} C_VEL
LIN {X 0,Y 192.744,Z 498.031,A -85,B 0,C 180,E1 -22280.349,E2 -22280.349} C_VEL
LIN {X 0,Y 190.407,Z 494.598,A -85,B 0,C 180,E1 -22281.414,E2 -22281.414} C_VEL
LIN {X 0,Y 189.802,Z 493.115,A -85,B 0,C 180,E1 -22281.776,E2 -22281.776} C_VEL
LIN {X 0,Y 188.959,Z 489.073,A -85,B 0,C 180,E1 -22286.089,E2 -22286.089} C_VEL
LIN {X 0,Y 187.944,Z 485.036,A -85,B 0,C 180,E1 -22290.914,E2 -22290.914} C_VEL
LIN {X 0,Y 187.168,Z 481.532,A -85,B 0,C 180,E1 -22295.604,E2 -22295.604} C_VEL
LIN {X 0,Y 186.366,Z 478.342,A -85,B 0,C 180,E1 -22300.512,E2 -22300.512} C_VEL
LIN {X 0,Y 185.741,Z 475.967,A -85,B 0,C 180,E1 -22305.202,E2 -22305.202} C_VEL
LIN {X 0,Y 185.934,Z 475.947,A -85,B 0,C 180,E1 -22309.328,E2 -22309.328} C_VEL
LIN {X 0,Y 185.961,Z 475.945,A -85,B 0,C 180,E1 -22313.49,E2 -22313.49} C_VEL
LIN {X 0,Y 186.22,Z 475.907,A -85,B 0,C 180,E1 -22317.837,E2 -22317.837} C_VEL
LIN {X 0,Y 186.4,Z 475.892,A -85,B 0,C 180,E1 -22320,E2 -22320} C_VEL
LIN {X 0,Y 185.916,Z 475.916,A -85,B 0,C 180,E1 -22324.336,E2 -22324.336} C_VEL
LIN {X 0,Y 186.019,Z 475.917,A -85,B 0,C 180,E1 -22328.692,E2 -22328.692} C_VEL
LIN {X 0,Y 185.76,Z 475.956,A -85,B 0,C 180,E1 -22333.121,E2 -22333.121} C_VEL
LIN {X 0,Y 185.666,Z 475.957,A -85,B 0,C 180,E1 -22338.868,E2 -22338.868} C_VEL
LIN {X 0,Y 185.606,Z 476.043,A -85,B 0,C 180,E1 -22341.374,E2 -22341.374} C_VEL
LIN {X 0,Y 186.88,Z 479.843,A -85,B 0,C 180,E1 -22346.826,E2 -22346.826} C_VEL
LIN {X 0,Y 187.67,Z 481.749,A -85,B 0,C 180,E1 -22349.133,E2 -22349.133} C_VEL
LIN {X 0,Y 189.226,Z 486.425,A -85,B 0,C 180,E1 -22353.856,E2 -22353.856} C_VEL
LIN {X 0,Y 190.777,Z 490.565,A -85,B 0,C 180,E1 -22357.433,E2 -22357.433} C_VEL
LIN {X 0,Y 191.488,Z 492.752,A -85,B 0,C 180,E1 -22359.061,E2 -22359.061} C_VEL
LIN {X 0,Y 194.753,Z 497.668,A -85,B 0,C 180,E1 -22360.508,E2 -22360.508} C_VEL
LIN {X 0,Y 200.317,Z 507.693,A -85,B 0,C 180,E1 -22362.988,E2 -22362.988} C_VEL
LIN {X 0,Y 205.685,Z 519.205,A -85,B 0,C 180,E1 -22365.589,E2 -22365.589} C_VEL
LIN {X 0,Y 208.82,Z 527.876,A -85,B 0,C 180,E1 -22367.41,E2 -22367.41} C_VEL
LIN {X 0,Y 209.921,Z 539.517,A -85,B 0,C 180,E1 -22369.29,E2 -22369.29} C_VEL
LIN {X 0,Y 209.782,Z 552.248,A -85,B 0,C 180,E1 -22371.45,E2 -22371.45} C_VEL
LIN {X 0,Y 209.033,Z 562.338,A -85,B 0,C 180,E1 -22373.364,E2 -22373.364} C_VEL
LIN {X 0,Y 205.524,Z 573.59,A -85,B 0,C 180,E1 -22375.427,E2 -22375.427} C_VEL
LIN {X 0,Y 201.502,Z 584.373,A -85,B 0,C 180,E1 -22377.87,E2 -22377.87} C_VEL
LIN {X 0,Y 197.315,Z 594.276,A -85,B 0,C 180,E1 -22380.679,E2 -22380.679} C_VEL
LIN {X 0,Y 193.209,Z 603.712,A -85,B 0,C 180,E1 -22384.122,E2 -22384.122} C_VEL
LIN {X 0,Y 190.244,Z 610.326,A -85,B 0,C 180,E1 -22387.181,E2 -22387.181} C_VEL
LIN {X 0,Y 187.887,Z 615.806,A -85,B 0,C 180,E1 -22390.33,E2 -22390.33} C_VEL
LIN {X 0,Y 185.506,Z 621.344,A -85,B 0,C 180,E1 -22394.442,E2 -22394.442} C_VEL
LIN {X 0,Y 184.077,Z 623.228,A -85,B 0,C 180,E1 -22396.124,E2 -22396.124} C_VEL
LIN {X 0,Y 180.349,Z 625.811,A -85,B 0,C 180,E1 -22398.895,E2 -22398.895} C_VEL
LIN {X 0,Y 177.488,Z 627.415,A -85,B 0,C 180,E1 -22401.218,E2 -22401.218} C_VEL
LIN {X 0,Y 176.216,Z 628.348,A -85,B 0,C 180,E1 -22403.071,E2 -22403.071} C_VEL
LIN {X 0,Y 176.068,Z 628.589,A -85,B 0,C 180,E1 -22403.707,E2 -22403.707} C_VEL
LIN {X 0,Y 175.949,Z 629.721,A -85,B 0,C 180,E1 -22407.714,E2 -22407.714} C_VEL
LIN {X 0,Y 175.996,Z 629.884,A -85,B 0,C 180,E1 -22410.003,E2 -22410.003} C_VEL
LIN {X 0,Y 175.979,Z 629.193,A -85,B 0,C 180,E1 -22414.584,E2 -22414.584} C_VEL
LIN {X 0,Y 176.446,Z 627.146,A -85,B 0,C 180,E1 -22419.17,E2 -22419.17} C_VEL
LIN {X 0,Y 177.62,Z 623.697,A -85,B 0,C 180,E1 -22423.736,E2 -22423.736} C_VEL
LIN {X 0,Y 179.827,Z 618.745,A -85,B 0,C 180,E1 -22428.222,E2 -22428.222} C_VEL
LIN {X 0,Y 181.706,Z 614.997,A -85,B 0,C 180,E1 -22430.966,E2 -22430.966} C_VEL
LIN {X 0,Y 185.177,Z 613.99,A -85,B 0,C 180,E1 -22434.678,E2 -22434.678} C_VEL
LIN {X 0,Y 190.416,Z 611.909,A -85,B 0,C 180,E1 -22438.676,E2 -22438.676} C_VEL
LIN {X 0,Y 196.705,Z 608.88,A -85,B 0,C 180,E1 -22442.41,E2 -22442.41} C_VEL
LIN {X 0,Y 206.121,Z 603.742,A -85,B 0,C 180,E1 -22446.636,E2 -22446.636} C_VEL
LIN {X 0,Y 217.11,Z 596.936,A -85,B 0,C 180,E1 -22450.349,E2 -22450.349} C_VEL
LIN {X 0,Y 226.855,Z 590.258,A -85,B 0,C 180,E1 -22452.968,E2 -22452.968} C_VEL
LIN {X 0,Y 229.409,Z 588.391,A -85,B 0,C 180,E1 -22453.577,E2 -22453.577} C_VEL
LIN {X 0,Y 231.236,Z 586.833,A -85,B 0,C 180,E1 -22454.353,E2 -22454.353} C_VEL
LIN {X 0,Y 231.614,Z 586.09,A -85,B 0,C 180,E1 -22455.741,E2 -22455.741} C_VEL
LIN {X 0,Y 231.333,Z 585.797,A -85,B 0,C 180,E1 -22458.059,E2 -22458.059} C_VEL
LIN {X 0,Y 230.034,Z 586.571,A -85,B 0,C 180,E1 -22460.09,E2 -22460.09} C_VEL
LIN {X 0,Y 228.391,Z 587.688,A -85,B 0,C 180,E1 -22460.889,E2 -22460.889} C_VEL
LIN {X 0,Y 218.601,Z 593.518,A -85,B 0,C 180,E1 -22463.618,E2 -22463.618} C_VEL
LIN {X 0,Y 212.147,Z 596.865,A -85,B 0,C 180,E1 -22465.725,E2 -22465.725} C_VEL
LIN {X 0,Y 203.951,Z 600.486,A -85,B 0,C 180,E1 -22468.876,E2 -22468.876} C_VEL
LIN {X 0,Y 196.726,Z 602.935,A -85,B 0,C 180,E1 -22472.327,E2 -22472.327} C_VEL
LIN {X 0,Y 190.637,Z 604.253,A -85,B 0,C 180,E1 -22476.076,E2 -22476.076} C_VEL
LIN {X 0,Y 185.456,Z 604.459,A -85,B 0,C 180,E1 -22480.059,E2 -22480.059} C_VEL
LIN {X 0,Y 181.728,Z 603.472,A -85,B 0,C 180,E1 -22484.294,E2 -22484.294} C_VEL
LIN {X 0,Y 178.878,Z 601.294,A -85,B 0,C 180,E1 -22488.671,E2 -22488.671} C_VEL
LIN {X 0,Y 177.164,Z 597.857,A -85,B 0,C 180,E1 -22493.165,E2 -22493.165} C_VEL
LIN {X 0,Y 176.587,Z 593.057,A -85,B 0,C 180,E1 -22497.719,E2 -22497.719} C_VEL
LIN {X 0,Y 176.458,Z 588.4,A -85,B 0,C 180,E1 -22501.141,E2 -22501.141} C_VEL
LIN {X 0,Y 176.612,Z 581.276,A -85,B 0,C 180,E1 -22505.324,E2 -22505.324} C_VEL
LIN {X 0,Y 177.169,Z 573.273,A -85,B 0,C 180,E1 -22509.13,E2 -22509.13} C_VEL
LIN {X 0,Y 178.077,Z 564.485,A -85,B 0,C 180,E1 -22512.537,E2 -22512.537} C_VEL
LIN {X 0,Y 179.456,Z 553.954,A -85,B 0,C 180,E1 -22515.911,E2 -22515.911} C_VEL
LIN {X 0,Y 181.322,Z 541.182,A -85,B 0,C 180,E1 -22519.236,E2 -22519.236} C_VEL
LIN {X 0,Y 183.062,Z 528.031,A -85,B 0,C 180,E1 -22521.982,E2 -22521.982} C_VEL
LIN {X 0,Y 181.187,Z 514.501,A -85,B 0,C 180,E1 -22524.339,E2 -22524.339} C_VEL
LIN {X 0,Y 178.948,Z 498.709,A -85,B 0,C 180,E1 -22526.563,E2 -22526.563} C_VEL
LIN {X 0,Y 177.893,Z 488.345,A -85,B 0,C 180,E1 -22527.771,E2 -22527.771} C_VEL
LIN {X 0,Y 179.35,Z 490.044,A -85,B 0,C 180,E1 -22530.625,E2 -22530.625} C_VEL
LIN {X 0,Y 181.731,Z 493.142,A -85,B 0,C 180,E1 -22535.155,E2 -22535.155} C_VEL
LIN {X 0,Y 184.148,Z 496.656,A -85,B 0,C 180,E1 -22536.437,E2 -22536.437} C_VEL
LIN {X 0,Y 186.578,Z 499.299,A -85,B 0,C 180,E1 -22537.622,E2 -22537.622} C_VEL
LIN {X 0,Y 189.179,Z 503.485,A -85,B 0,C 180,E1 -22538.95,E2 -22538.95} C_VEL
LIN {X 0,Y 193.444,Z 511.25,A -85,B 0,C 180,E1 -22541.186,E2 -22541.186} C_VEL
LIN {X 0,Y 197.823,Z 520.608,A -85,B 0,C 180,E1 -22543.674,E2 -22543.674} C_VEL
LIN {X 0,Y 200.155,Z 529.495,A -85,B 0,C 180,E1 -22545.561,E2 -22545.561} C_VEL
LIN {X 0,Y 202.085,Z 541.626,A -85,B 0,C 180,E1 -22548.073,E2 -22548.073} C_VEL
LIN {X 0,Y 202.81,Z 552.639,A -85,B 0,C 180,E1 -22550.422,E2 -22550.422} C_VEL
LIN {X 0,Y 202.646,Z 563.556,A -85,B 0,C 180,E1 -22552.908,E2 -22552.908} C_VEL
LIN {X 0,Y 201.583,Z 567.316,A -85,B 0,C 180,E1 -22553.649,E2 -22553.649} C_VEL
LIN {X 0,Y 197.543,Z 577.962,A -85,B 0,C 180,E1 -22555.918,E2 -22555.918} C_VEL
LIN {X 0,Y 193.766,Z 586.888,A -85,B 0,C 180,E1 -22558.267,E2 -22558.267} C_VEL
LIN {X 0,Y 189.845,Z 595.844,A -85,B 0,C 180,E1 -22561.23,E2 -22561.23} C_VEL
LIN {X 0,Y 185.687,Z 604.4,A -85,B 0,C 180,E1 -22564.796,E2 -22564.796} C_VEL
LIN {X 0,Y 182.526,Z 611.294,A -85,B 0,C 180,E1 -22568.541,E2 -22568.541} C_VEL
LIN {X 0,Y 180.256,Z 616.063,A -85,B 0,C 180,E1 -22571.823,E2 -22571.823} C_VEL
LIN {X 0,Y 177.971,Z 620.975,A -85,B 0,C 180,E1 -22576.291,E2 -22576.291} C_VEL
LIN {X 0,Y 176.628,Z 624.396,A -85,B 0,C 180,E1 -22580.839,E2 -22580.839} C_VEL
LIN {X 0,Y 176.013,Z 626.428,A -85,B 0,C 180,E1 -22585.417,E2 -22585.417} C_VEL
LIN {X 0,Y 175.982,Z 627.122,A -85,B 0,C 180,E1 -22589.997,E2 -22589.997} C_VEL
LIN {X 0,Y 176.012,Z 626.483,A -85,B 0,C 180,E1 -22594.577,E2 -22594.577} C_VEL
LIN {X 0,Y 176.623,Z 624.498,A -85,B 0,C 180,E1 -22599.155,E2 -22599.155} C_VEL
LIN {X 0,Y 177.932,Z 621.123,A -85,B 0,C 180,E1 -22603.706,E2 -22603.706} C_VEL
LIN {X 0,Y 180.173,Z 616.254,A -85,B 0,C 180,E1 -22608.18,E2 -22608.18} C_VEL
LIN {X 0,Y 182.475,Z 611.537,A -85,B 0,C 180,E1 -22611.459,E2 -22611.459} C_VEL
LIN {X 0,Y 185.668,Z 604.701,A -85,B 0,C 180,E1 -22615.201,E2 -22615.201} C_VEL
LIN {X 0,Y 189.75,Z 596.207,A -85,B 0,C 180,E1 -22618.78,E2 -22618.78} C_VEL
LIN {X 0,Y 193.701,Z 587.323,A -85,B 0,C 180,E1 -22621.739,E2 -22621.739} C_VEL
LIN {X 0,Y 198.257,Z 576.559,A -85,B 0,C 180,E1 -22624.551,E2 -22624.551} C_VEL
LIN {X 0,Y 202.29,Z 565.654,A -85,B 0,C 180,E1 -22626.809,E2 -22626.809} C_VEL
LIN {X 0,Y 202.756,Z 562.853,A -85,B 0,C 180,E1 -22627.403,E2 -22627.403} C_VEL
LIN {X 0,Y 202.862,Z 551.047,A -85,B 0,C 180,E1 -22630.065,E2 -22630.065} C_VEL
LIN {X 0,Y 201.98,Z 540.168,A -85,B 0,C 180,E1 -22632.378,E2 -22632.378} C_VEL
LIN {X 0,Y 199.865,Z 528.041,A -85,B 0,C 180,E1 -22634.901,E2 -22634.901} C_VEL
LIN {X 0,Y 197.94,Z 520.81,A -85,B 0,C 180,E1 -22636.446,E2 -22636.446} C_VEL
LIN {X 0,Y 194.042,Z 512.273,A -85,B 0,C 180,E1 -22638.69,E2 -22638.69} C_VEL
LIN {X 0,Y 191.012,Z 506.737,A -85,B 0,C 180,E1 -22640.286,E2 -22640.286} C_VEL
LIN {X 0,Y 189.102,Z 503.331,A -85,B 0,C 180,E1 -22641.293,E2 -22641.293} C_VEL
LIN {X 0,Y 186.733,Z 499.527,A -85,B 0,C 180,E1 -22642.507,E2 -22642.507} C_VEL
LIN {X 0,Y 185.796,Z 498.118,A -85,B 0,C 180,E1 -22642.996,E2 -22642.996} C_VEL
LIN {X 0,Y 183.239,Z 494.376,A -85,B 0,C 180,E1 -22644.321,E2 -22644.321} C_VEL
LIN {X 0,Y 182.717,Z 493.126,A -85,B 0,C 180,E1 -22644.654,E2 -22644.654} C_VEL
LIN {X 0,Y 182.029,Z 490.197,A -85,B 0,C 180,E1 -22648.141,E2 -22648.141} C_VEL
LIN {X 0,Y 181.099,Z 486.298,A -85,B 0,C 180,E1 -22653.191,E2 -22653.191} C_VEL
LIN {X 0,Y 180.478,Z 483.686,A -85,B 0,C 180,E1 -22657.082,E2 -22657.082} C_VEL
LIN {X 0,Y 179.817,Z 480.906,A -85,B 0,C 180,E1 -22661.779,E2 -22661.779} C_VEL
LIN {X 0,Y 179.195,Z 478.732,A -85,B 0,C 180,E1 -22666.389,E2 -22666.389} C_VEL
LIN {X 0,Y 178.969,Z 476.811,A -85,B 0,C 180,E1 -22670.963,E2 -22670.963} C_VEL
LIN {X 0,Y 179.164,Z 476.786,A -85,B 0,C 180,E1 -22677.752,E2 -22677.752} C_VEL
LIN {X 0,Y 179.363,Z 476.769,A -85,B 0,C 180,E1 -22680,E2 -22680} C_VEL
LIN {X 0,Y 178.865,Z 476.795,A -85,B 0,C 180,E1 -22684.507,E2 -22684.507} C_VEL
LIN {X 0,Y 178.969,Z 476.79,A -85,B 0,C 180,E1 -22689.037,E2 -22689.037} C_VEL
LIN {X 0,Y 178.668,Z 476.855,A -85,B 0,C 180,E1 -22694.232,E2 -22694.232} C_VEL
LIN {X 0,Y 179.505,Z 479.658,A -85,B 0,C 180,E1 -22700.632,E2 -22700.632} C_VEL
LIN {X 0,Y 180.882,Z 483.615,A -85,B 0,C 180,E1 -22706.673,E2 -22706.673} C_VEL
LIN {X 0,Y 181.953,Z 486.569,A -85,B 0,C 180,E1 -22710.141,E2 -22710.141} C_VEL
LIN {X 0,Y 183.661,Z 491.47,A -85,B 0,C 180,E1 -22715.029,E2 -22715.029} C_VEL
LIN {X 0,Y 184.223,Z 492.864,A -85,B 0,C 180,E1 -22716.184,E2 -22716.184} C_VEL
LIN {X 0,Y 187.311,Z 497.375,A -85,B 0,C 180,E1 -22717.738,E2 -22717.738} C_VEL
LIN {X 0,Y 188.855,Z 499.527,A -85,B 0,C 180,E1 -22718.474,E2 -22718.474} C_VEL
LIN {X 0,Y 191.771,Z 504.188,A -85,B 0,C 180,E1 -22719.89,E2 -22719.89} C_VEL
LIN {X 0,Y 196.117,Z 512.427,A -85,B 0,C 180,E1 -22722.067,E2 -22722.067} C_VEL
LIN {X 0,Y 200.836,Z 523.349,A -85,B 0,C 180,E1 -22724.707,E2 -22724.707} C_VEL
LIN {X 0,Y 203.525,Z 531.274,A -85,B 0,C 180,E1 -22726.482,E2 -22726.482} C_VEL
LIN {X 0,Y 204.246,Z 541.68,A -85,B 0,C 180,E1 -22728.275,E2 -22728.275} C_VEL
LIN {X 0,Y 203.875,Z 554.122,A -85,B 0,C 180,E1 -22730.506,E2 -22730.506} C_VEL
LIN {X 0,Y 202.977,Z 563.595,A -85,B 0,C 180,E1 -22732.395,E2 -22732.395} C_VEL
LIN {X 0,Y 199.021,Z 575.322,A -85,B 0,C 180,E1 -22734.646,E2 -22734.646} C_VEL
LIN {X 0,Y 194.724,Z 586.097,A -85,B 0,C 180,E1 -22737.226,E2 -22737.226} C_VEL
LIN {X 0,Y 190.495,Z 595.705,A -85,B 0,C 180,E1 -22740.132,E2 -22740.132} C_VEL
LIN {X 0,Y 186.804,Z 603.661,A -85,B 0,C 180,E1 -22743.166,E2 -22743.166} C_VEL
LIN {X 0,Y 183.69,Z 610.274,A -85,B 0,C 180,E1 -22746.318,E2 -22746.318} C_VEL
LIN {X 0,Y 181.174,Z 615.753,A -85,B 0,C 180,E1 -22749.57,E2 -22749.57} C_VEL
LIN {X 0,Y 179.175,Z 620.244,A -85,B 0,C 180,E1 -22752.895,E2 -22752.895} C_VEL
LIN {X 0,Y 177.622,Z 623.763,A -85,B 0,C 180,E1 -22756.27,E2 -22756.27} C_VEL
LIN {X 0,Y 176.443,Z 627.193,A -85,B 0,C 180,E1 -22760.835,E2 -22760.835} C_VEL
LIN {X 0,Y 176.068,Z 628.589,A -85,B 0,C 180,E1 -22763.707,E2 -22763.707} C_VEL
LIN {X 0,Y 175.257,Z 629.275,A -85,B 0,C 180,E1 -22765.606,E2 -22765.606} C_VEL
LIN {X 0,Y 173.604,Z 629.663,A -85,B 0,C 180,E1 -22767.48,E2 -22767.48} C_VEL
LIN {X 0,Y 169.894,Z 629.753,A -85,B 0,C 180,E1 -22771.294,E2 -22771.294} C_VEL
LIN {X 0,Y 168.904,Z 629.471,A -85,B 0,C 180,E1 -22773.291,E2 -22773.291} C_VEL
LIN {X 0,Y 168.841,Z 629.313,A -85,B 0,C 180,E1 -22773.967,E2 -22773.967} C_VEL
LIN {X 0,Y 169.07,Z 628.284,A -85,B 0,C 180,E1 -22777.167,E2 -22777.167} C_VEL
LIN {X 0,Y 169.956,Z 625.546,A -85,B 0,C 180,E1 -22781.935,E2 -22781.935} C_VEL
LIN {X 0,Y 171.713,Z 621.362,A -85,B 0,C 180,E1 -22786.652,E2 -22786.652} C_VEL
LIN {X 0,Y 174.619,Z 615.603,A -85,B 0,C 180,E1 -22791.24,E2 -22791.24} C_VEL
LIN {X 0,Y 175.274,Z 614.571,A -85,B 0,C 180,E1 -22792.084,E2 -22792.084} C_VEL
LIN {X 0,Y 178.722,Z 613.854,A -85,B 0,C 180,E1 -22795.633,E2 -22795.633} C_VEL
LIN {X 0,Y 184.214,Z 612.154,A -85,B 0,C 180,E1 -22799.736,E2 -22799.736} C_VEL
LIN {X 0,Y 190.791,Z 609.496,A -85,B 0,C 180,E1 -22803.544,E2 -22803.544} C_VEL
LIN {X 0,Y 200.546,Z 604.872,A -85,B 0,C 180,E1 -22807.83,E2 -22807.83} C_VEL
LIN {X 0,Y 209.516,Z 600.048,A -85,B 0,C 180,E1 -22810.855,E2 -22810.855} C_VEL
LIN {X 0,Y 219.339,Z 594.18,A -85,B 0,C 180,E1 -22813.546,E2 -22813.546} C_VEL
LIN {X 0,Y 224.521,Z 590.817,A -85,B 0,C 180,E1 -22814.776,E2 -22814.776} C_VEL
LIN {X 0,Y 225.579,Z 589.867,A -85,B 0,C 180,E1 -22815.775,E2 -22815.775} C_VEL
LIN {X 0,Y 225.566,Z 589.609,A -85,B 0,C 180,E1 -22816.728,E2 -22816.728} C_VEL
LIN {X 0,Y 224.659,Z 589.859,A -85,B 0,C 180,E1 -22818.933,E2 -22818.933} C_VEL
LIN {X 0,Y 223.224,Z 590.62,A -85,B 0,C 180,E1 -22819.803,E2 -22819.803} C_VEL
LIN {X 0,Y 213.469,Z 595.757,A -85,B 0,C 180,E1 -22822.448,E2 -22822.448} C_VEL
LIN {X 0,Y 206.521,Z 598.909,A -85,B 0,C 180,E1 -22824.654,E2 -22824.654} C_VEL
LIN {X 0,Y 198.047,Z 602.051,A -85,B 0,C 180,E1 -22827.839,E2 -22827.839} C_VEL
LIN {X 0,Y 190.552,Z 604.102,A -85,B 0,C 180,E1 -22831.349,E2 -22831.349} C_VEL
LIN {X 0,Y 184.227,Z 605.026,A -85,B 0,C 180,E1 -22835.189,E2 -22835.189} C_VEL
LIN {X 0,Y 178.826,Z 604.854,A -85,B 0,C 180,E1 -22839.286,E2 -22839.286} C_VEL
LIN {X 0,Y 174.908,Z 603.517,A -85,B 0,C 180,E1 -22843.664,E2 -22843.664} C_VEL
LIN {X 0,Y 171.94,Z 601,A -85,B 0,C 180,E1 -22848.207,E2 -22848.207} C_VEL
LIN {X 0,Y 170.168,Z 597.247,A -85,B 0,C 180,E1 -22852.883,E2 -22852.883} C_VEL
LIN {X 0,Y 169.549,Z 592.111,A -85,B 0,C 180,E1 -22857.625,E2 -22857.625} C_VEL
LIN {X 0,Y 169.451,Z 587.227,A -85,B 0,C 180,E1 -22861.188,E2 -22861.188} C_VEL
LIN {X 0,Y 169.568,Z 581.264,A -85,B 0,C 180,E1 -22864.755,E2 -22864.755} C_VEL
LIN {X 0,Y 170.109,Z 572.754,A -85,B 0,C 180,E1 -22868.913,E2 -22868.913} C_VEL
LIN {X 0,Y 170.997,Z 563.946,A -85,B 0,C 180,E1 -22872.461,E2 -22872.461} C_VEL
LIN {X 0,Y 172.397,Z 553.285,A -85,B 0,C 180,E1 -22875.973,E2 -22875.973} C_VEL
LIN {X 0,Y 174.123,Z 541.505,A -85,B 0,C 180,E1 -22879.144,E2 -22879.144} C_VEL
LIN {X 0,Y 175.884,Z 529.09,A -85,B 0,C 180,E1 -22881.861,E2 -22881.861} C_VEL
LIN {X 0,Y 175.023,Z 521.638,A -85,B 0,C 180,E1 -22883.281,E2 -22883.281} C_VEL
LIN {X 0,Y 173.105,Z 508.489,A -85,B 0,C 180,E1 -22885.46,E2 -22885.46} C_VEL
LIN {X 0,Y 171.218,Z 493.255,A -85,B 0,C 180,E1 -22887.502,E2 -22887.502} C_VEL
LIN {X 0,Y 171.049,Z 491.534,A -85,B 0,C 180,E1 -22887.698,E2 -22887.698} C_VEL
LIN {X 0,Y 172.213,Z 492.267,A -85,B 0,C 180,E1 -22889.322,E2 -22889.322} C_VEL
LIN {X 0,Y 173.094,Z 493.352,A -85,B 0,C 180,E1 -22890.888,E2 -22890.888} C_VEL
LIN {X 0,Y 175.677,Z 496.685,A -85,B 0,C 180,E1 -22892.519,E2 -22892.519} C_VEL
LIN {X 0,Y 179.198,Z 499.78,A -85,B 0,C 180,E1 -22894.49,E2 -22894.49} C_VEL
LIN {X 0,Y 182.802,Z 504.361,A -85,B 0,C 180,E1 -22896.482,E2 -22896.482} C_VEL
LIN {X 0,Y 186.315,Z 510.374,A -85,B 0,C 180,E1 -22898.52,E2 -22898.52} C_VEL
LIN {X 0,Y 190.436,Z 518.588,A -85,B 0,C 180,E1 -22901.012,E2 -22901.012} C_VEL
LIN {X 0,Y 193.653,Z 526.833,A -85,B 0,C 180,E1 -22903.237,E2 -22903.237} C_VEL
LIN {X 0,Y 195.615,Z 537.449,A -85,B 0,C 180,E1 -22905.564,E2 -22905.564} C_VEL
LIN {X 0,Y 196.716,Z 547.659,A -85,B 0,C 180,E1 -22907.845,E2 -22907.845} C_VEL
LIN {X 0,Y 196.886,Z 558.528,A -85,B 0,C 180,E1 -22910.347,E2 -22910.347} C_VEL
LIN {X 0,Y 196.376,Z 566.11,A -85,B 0,C 180,E1 -22912.171,E2 -22912.171} C_VEL
LIN {X 0,Y 192.518,Z 576.084,A -85,B 0,C 180,E1 -22914.258,E2 -22914.258} C_VEL
LIN {X 0,Y 187.746,Z 586.941,A -85,B 0,C 180,E1 -22917.124,E2 -22917.124} C_VEL
LIN {X 0,Y 183.638,Z 595.899,A -85,B 0,C 180,E1 -22920.161,E2 -22920.161} C_VEL
LIN {X 0,Y 179.256,Z 604.455,A -85,B 0,C 180,E1 -22923.825,E2 -22923.825} C_VEL
LIN {X 0,Y 175.877,Z 611.35,A -85,B 0,C 180,E1 -22927.687,E2 -22927.687} C_VEL
LIN {X 0,Y 173.487,Z 616.119,A -85,B 0,C 180,E1 -22931.087,E2 -22931.087} C_VEL
LIN {X 0,Y 171.065,Z 621.032,A -85,B 0,C 180,E1 -22935.726,E2 -22935.726} C_VEL
LIN {X 0,Y 169.616,Z 624.452,A -85,B 0,C 180,E1 -22940.457,E2 -22940.457} C_VEL
LIN {X 0,Y 168.938,Z 626.484,A -85,B 0,C 180,E1 -22945.224,E2 -22945.224} C_VEL
LIN {X 0,Y 168.881,Z 627.178,A -85,B 0,C 180,E1 -22949.997,E2 -22949.997} C_VEL
LIN {X 0,Y 168.937,Z 626.539,A -85,B 0,C 180,E1 -22954.77,E2 -22954.77} C_VEL
LIN {X 0,Y 169.611,Z 624.553,A -85,B 0,C 180,E1 -22959.537,E2 -22959.537} C_VEL
LIN {X 0,Y 171.02,Z 621.177,A -85,B 0,C 180,E1 -22964.271,E2 -22964.271} C_VEL
LIN {X 0,Y 172.68,Z 617.706,A -85,B 0,C 180,E1 -22967.77,E2 -22967.77} C_VEL
LIN {X 0,Y 175.016,Z 613.27,A -85,B 0,C 180,E1 -22971.183,E2 -22971.183} C_VEL
LIN {X 0,Y 177.874,Z 607.415,A -85,B 0,C 180,E1 -22974.788,E2 -22974.788} C_VEL
LIN {X 0,Y 181.572,Z 600.122,A -85,B 0,C 180,E1 -22978.301,E2 -22978.301} C_VEL
LIN {X 0,Y 185.535,Z 592.02,A -85,B 0,C 180,E1 -22981.385,E2 -22981.385} C_VEL
LIN {X 0,Y 190.003,Z 582.253,A -85,B 0,C 180,E1 -22984.335,E2 -22984.335} C_VEL
LIN {X 0,Y 194.527,Z 571.393,A -85,B 0,C 180,E1 -22986.912,E2 -22986.912} C_VEL
LIN {X 0,Y 196.614,Z 565.349,A -85,B 0,C 180,E1 -22988.15,E2 -22988.15} C_VEL
LIN {X 0,Y 197.006,Z 554.435,A -85,B 0,C 180,E1 -22990.774,E2 -22990.774} C_VEL
LIN {X 0,Y 196.503,Z 544.085,A -85,B 0,C 180,E1 -22993.109,E2 -22993.109} C_VEL
LIN {X 0,Y 195.029,Z 533.275,A -85,B 0,C 180,E1 -22995.501,E2 -22995.501} C_VEL
LIN {X 0,Y 193.543,Z 526.135,A -85,B 0,C 180,E1 -22997.089,E2 -22997.089} C_VEL
LIN {X 0,Y 190.11,Z 517.613,A -85,B 0,C 180,E1 -22999.427,E2 -22999.427} C_VEL
LIN {X 0,Y 185.563,Z 508.861,A -85,B 0,C 180,E1 -23002.135,E2 -23002.135} C_VEL
LIN {X 0,Y 182.359,Z 503.511,A -85,B 0,C 180,E1 -23003.997,E2 -23003.997} C_VEL
LIN {X 0,Y 179.827,Z 499.402,A -85,B 0,C 180,E1 -23005.48,E2 -23005.48} C_VEL
LIN {X 0,Y 176.418,Z 494.963,A -85,B 0,C 180,E1 -23007.478,E2 -23007.478} C_VEL
LIN {X 0,Y 175.557,Z 493.127,A -85,B 0,C 180,E1 -23008.088,E2 -23008.088} C_VEL
LIN {X 0,Y 174.605,Z 489.008,A -85,B 0,C 180,E1 -23013.72,E2 -23013.72} C_VEL
LIN {X 0,Y 173.891,Z 485.89,A -85,B 0,C 180,E1 -23018.669,E2 -23018.669} C_VEL
LIN {X 0,Y 173.295,Z 483.352,A -85,B 0,C 180,E1 -23023.508,E2 -23023.508} C_VEL
LIN {X 0,Y 172.824,Z 480.548,A -85,B 0,C 180,E1 -23030.638,E2 -23030.638} C_VEL
LIN {X 0,Y 172.354,Z 478.887,A -85,B 0,C 180,E1 -23037.663,E2 -23037.663} C_VEL
LIN {X 0,Y 172.474,Z 478.517,A -85,B 0,C 180,E1 -23040,E2 -23040} C_VEL
LIN {X 0,Y 172.063,Z 478.811,A -85,B 0,C 180,E1 -23044.686,E2 -23044.686} C_VEL
LIN {X 0,Y 172.317,Z 479.347,A -85,B 0,C 180,E1 -23049.389,E2 -23049.389} C_VEL
LIN {X 0,Y 172.66,Z 480.632,A -85,B 0,C 180,E1 -23054.136,E2 -23054.136} C_VEL
LIN {X 0,Y 173.174,Z 482.677,A -85,B 0,C 180,E1 -23058.945,E2 -23058.945} C_VEL
LIN {X 0,Y 174.148,Z 485.479,A -85,B 0,C 180,E1 -23063.801,E2 -23063.801} C_VEL
LIN {X 0,Y 175.568,Z 489.054,A -85,B 0,C 180,E1 -23068.709,E2 -23068.709} C_VEL
LIN {X 0,Y 176.888,Z 493.002,A -85,B 0,C 180,E1 -23072.795,E2 -23072.795} C_VEL
LIN {X 0,Y 179.828,Z 497.225,A -85,B 0,C 180,E1 -23074.519,E2 -23074.519} C_VEL
LIN {X 0,Y 181.507,Z 499.202,A -85,B 0,C 180,E1 -23075.422,E2 -23075.422} C_VEL
LIN {X 0,Y 185.631,Z 505.301,A -85,B 0,C 180,E1 -23077.646,E2 -23077.646} C_VEL
LIN {X 0,Y 188.525,Z 510.356,A -85,B 0,C 180,E1 -23079.24,E2 -23079.24} C_VEL
LIN {X 0,Y 193.458,Z 520.919,A -85,B 0,C 180,E1 -23082.139,E2 -23082.139} C_VEL
LIN {X 0,Y 197.331,Z 531.419,A -85,B 0,C 180,E1 -23084.772,E2 -23084.772} C_VEL
LIN {X 0,Y 198.217,Z 534.716,A -85,B 0,C 180,E1 -23085.539,E2 -23085.539} C_VEL
LIN {X 0,Y 198.617,Z 545.593,A -85,B 0,C 180,E1 -23087.522,E2 -23087.522} C_VEL
LIN {X 0,Y 197.797,Z 557.638,A -85,B 0,C 180,E1 -23089.821,E2 -23089.821} C_VEL
LIN {X 0,Y 196.627,Z 566.116,A -85,B 0,C 180,E1 -23091.612,E2 -23091.612} C_VEL
LIN {X 0,Y 192.572,Z 577.109,A -85,B 0,C 180,E1 -23093.834,E2 -23093.834} C_VEL
LIN {X 0,Y 188,Z 587.82,A -85,B 0,C 180,E1 -23096.54,E2 -23096.54} C_VEL
LIN {X 0,Y 183.669,Z 597.119,A -85,B 0,C 180,E1 -23099.539,E2 -23099.539} C_VEL
LIN {X 0,Y 179.871,Z 604.832,A -85,B 0,C 180,E1 -23102.674,E2 -23102.674} C_VEL
LIN {X 0,Y 175.949,Z 612.588,A -85,B 0,C 180,E1 -23106.736,E2 -23106.736} C_VEL
LIN {X 0,Y 173.051,Z 618.775,A -85,B 0,C 180,E1 -23111.044,E2 -23111.044} C_VEL
LIN {X 0,Y 170.678,Z 623.708,A -85,B 0,C 180,E1 -23115.699,E2 -23115.699} C_VEL
LIN {X 0,Y 169.399,Z 627.137,A -85,B 0,C 180,E1 -23120.451,E2 -23120.451} C_VEL
LIN {X 0,Y 168.88,Z 629.162,A -85,B 0,C 180,E1 -23125.229,E2 -23125.229} C_VEL
LIN {X 0,Y 168.858,Z 629.665,A -85,B 0,C 180,E1 -23127.618,E2 -23127.618} C_VEL
LIN {X 0,Y 168.908,Z 629.829,A -85,B 0,C 180,E1 -23130.003,E2 -23130.003} C_VEL
LIN {X 0,Y 168.841,Z 629.313,A -85,B 0,C 180,E1 -23133.967,E2 -23133.967} C_VEL
LIN {X 0,Y 168.585,Z 628.973,A -85,B 0,C 180,E1 -23135.295,E2 -23135.295} C_VEL
LIN {X 0,Y 166.884,Z 628.009,A -85,B 0,C 180,E1 -23137.911,E2 -23137.911} C_VEL
LIN {X 0,Y 163.908,Z 625.872,A -85,B 0,C 180,E1 -23141.855,E2 -23141.855} C_VEL
LIN {X 0,Y 163.513,Z 624.202,A -85,B 0,C 180,E1 -23144.208,E2 -23144.208} C_VEL
LIN {X 0,Y 163.611,Z 623.881,A -85,B 0,C 180,E1 -23144.543,E2 -23144.543} C_VEL
LIN {X 0,Y 165.586,Z 620.052,A -85,B 0,C 180,E1 -23148.565,E2 -23148.565} C_VEL
LIN {X 0,Y 168.941,Z 614.057,A -85,B 0,C 180,E1 -23153.278,E2 -23153.278} C_VEL
LIN {X 0,Y 175.057,Z 613.045,A -85,B 0,C 180,E1 -23158.804,E2 -23158.804} C_VEL
LIN {X 0,Y 181.382,Z 611.227,A -85,B 0,C 180,E1 -23162.854,E2 -23162.854} C_VEL
LIN {X 0,Y 188.836,Z 608.526,A -85,B 0,C 180,E1 -23166.55,E2 -23166.55} C_VEL
LIN {X 0,Y 197.3,Z 604.875,A -85,B 0,C 180,E1 -23169.882,E2 -23169.882} C_VEL
LIN {X 0,Y 209.245,Z 598.98,A -85,B 0,C 180,E1 -23173.518,E2 -23173.518} C_VEL
LIN {X 0,Y 217.023,Z 594.666,A -85,B 0,C 180,E1 -23175.437,E2 -23175.437} C_VEL
LIN {X 0,Y 219.389,Z 593.266,A -85,B 0,C 180,E1 -23176.121,E2 -23176.121} C_VEL
LIN {X 0,Y 218.986,Z 593.142,A -85,B 0,C 180,E1 -23177.627,E2 -23177.627} C_VEL
LIN {X 0,Y 218.134,Z 593.458,A -85,B 0,C 180,E1 -23178.663,E2 -23178.663} C_VEL
LIN {X 0,Y 205.613,Z 599.074,A -85,B 0,C 180,E1 -23182.03,E2 -23182.03} C_VEL
LIN {X 0,Y 196.461,Z 602.306,A -85,B 0,C 180,E1 -23185.085,E2 -23185.085} C_VEL
LIN {X 0,Y 188.196,Z 604.452,A -85,B 0,C 180,E1 -23188.479,E2 -23188.479} C_VEL
LIN {X 0,Y 181.014,Z 605.535,A -85,B 0,C 180,E1 -23192.231,E2 -23192.231} C_VEL
LIN {X 0,Y 174.874,Z 605.536,A -85,B 0,C 180,E1 -23196.304,E2 -23196.304} C_VEL
LIN {X 0,Y 170.022,Z 604.422,A -85,B 0,C 180,E1 -23200.69,E2 -23200.69} C_VEL
LIN {X 0,Y 166.387,Z 602.169,A -85,B 0,C 180,E1 -23205.319,E2 -23205.319} C_VEL
LIN {X 0,Y 163.878,Z 598.729,A -85,B 0,C 180,E1 -23210.123,E2 -23210.123} C_VEL
LIN {X 0,Y 162.737,Z 594,A -85,B 0,C 180,E1 -23215.045,E2 -23215.045} C_VEL
LIN {X 0,Y 162.46,Z 589.474,A -85,B 0,C 180,E1 -23218.761,E2 -23218.761} C_VEL
LIN {X 0,Y 162.469,Z 582.963,A -85,B 0,C 180,E1 -23223.1,E2 -23223.1} C_VEL
LIN {X 0,Y 162.867,Z 574.869,A -85,B 0,C 180,E1 -23227.438,E2 -23227.438} C_VEL
LIN {X 0,Y 163.781,Z 564.828,A -85,B 0,C 180,E1 -23231.761,E2 -23231.761} C_VEL
LIN {X 0,Y 165.07,Z 554.387,A -85,B 0,C 180,E1 -23235.432,E2 -23235.432} C_VEL
LIN {X 0,Y 166.72,Z 542.926,A -85,B 0,C 180,E1 -23238.75,E2 -23238.75} C_VEL
LIN {X 0,Y 168.377,Z 531.626,A -85,B 0,C 180,E1 -23241.422,E2 -23241.422} C_VEL
LIN {X 0,Y 168.823,Z 528.801,A -85,B 0,C 180,E1 -23242.004,E2 -23242.004} C_VEL
LIN {X 0,Y 167.149,Z 516.358,A -85,B 0,C 180,E1 -23244.383,E2 -23244.383} C_VEL
LIN {X 0,Y 165.13,Z 502.115,A -85,B 0,C 180,E1 -23246.643,E2 -23246.643} C_VEL
LIN {X 0,Y 165.078,Z 501.625,A -85,B 0,C 180,E1 -23246.761,E2 -23246.761} C_VEL
LIN {X 0,Y 165.765,Z 502.83,A -85,B 0,C 180,E1 -23247.369,E2 -23247.369} C_VEL
LIN {X 0,Y 166.928,Z 502.577,A -85,B 0,C 180,E1 -23248.101,E2 -23248.101} C_VEL
LIN {X 0,Y 168.618,Z 500.382,A -85,B 0,C 180,E1 -23248.917,E2 -23248.917} C_VEL
LIN {X 0,Y 169.186,Z 499.334,A -85,B 0,C 180,E1 -23249.148,E2 -23249.148} C_VEL
LIN {X 0,Y 170.404,Z 499.445,A -85,B 0,C 180,E1 -23249.886,E2 -23249.886} C_VEL
LIN {X 0,Y 174.277,Z 503.998,A -85,B 0,C 180,E1 -23252.47,E2 -23252.47} C_VEL
LIN {X 0,Y 176.279,Z 505.794,A -85,B 0,C 180,E1 -23253.671,E2 -23253.671} C_VEL
LIN {X 0,Y 180.036,Z 511.084,A -85,B 0,C 180,E1 -23256.015,E2 -23256.015} C_VEL
LIN {X 0,Y 183.008,Z 516.741,A -85,B 0,C 180,E1 -23257.999,E2 -23257.999} C_VEL
LIN {X 0,Y 186.583,Z 524.739,A -85,B 0,C 180,E1 -23260.524,E2 -23260.524} C_VEL
LIN {X 0,Y 188.607,Z 530.266,A -85,B 0,C 180,E1 -23262.124,E2 -23262.124} C_VEL
LIN {X 0,Y 190.031,Z 538.935,A -85,B 0,C 180,E1 -23264.174,E2 -23264.174} C_VEL
LIN {X 0,Y 190.963,Z 548.445,A -85,B 0,C 180,E1 -23266.42,E2 -23266.42} C_VEL
LIN {X 0,Y 190.995,Z 559.982,A -85,B 0,C 180,E1 -23269.219,E2 -23269.219} C_VEL
LIN {X 0,Y 190.306,Z 567.413,A -85,B 0,C 180,E1 -23271.108,E2 -23271.108} C_VEL
LIN {X 0,Y 185.936,Z 578.064,A -85,B 0,C 180,E1 -23273.462,E2 -23273.462} C_VEL
LIN {X 0,Y 181.042,Z 588.598,A -85,B 0,C 180,E1 -23276.411,E2 -23276.411} C_VEL
LIN {X 0,Y 176.798,Z 597.289,A -85,B 0,C 180,E1 -23279.544,E2 -23279.544} C_VEL
LIN {X 0,Y 172.311,Z 605.612,A -85,B 0,C 180,E1 -23283.34,E2 -23283.34} C_VEL
LIN {X 0,Y 169.282,Z 611.405,A -85,B 0,C 180,E1 -23286.768,E2 -23286.768} C_VEL
LIN {X 0,Y 166.757,Z 616.175,A -85,B 0,C 180,E1 -23290.293,E2 -23290.293} C_VEL
LIN {X 0,Y 164.159,Z 621.088,A -85,B 0,C 180,E1 -23295.112,E2 -23295.112} C_VEL
LIN {X 0,Y 162.597,Z 624.508,A -85,B 0,C 180,E1 -23300.041,E2 -23300.041} C_VEL
LIN {X 0,Y 161.859,Z 626.54,A -85,B 0,C 180,E1 -23305.015,E2 -23305.015} C_VEL
LIN {X 0,Y 161.78,Z 627.233,A -85,B 0,C 180,E1 -23309.997,E2 -23309.997} C_VEL
LIN {X 0,Y 161.858,Z 626.594,A -85,B 0,C 180,E1 -23314.979,E2 -23314.979} C_VEL
LIN {X 0,Y 162.591,Z 624.608,A -85,B 0,C 180,E1 -23319.953,E2 -23319.953} C_VEL
LIN {X 0,Y 164.109,Z 621.232,A -85,B 0,C 180,E1 -23324.886,E2 -23324.886} C_VEL
LIN {X 0,Y 165.913,Z 617.76,A -85,B 0,C 180,E1 -23328.52,E2 -23328.52} C_VEL
LIN {X 0,Y 168.363,Z 613.324,A -85,B 0,C 180,E1 -23332.063,E2 -23332.063} C_VEL
LIN {X 0,Y 171.285,Z 607.719,A -85,B 0,C 180,E1 -23335.645,E2 -23335.645} C_VEL
LIN {X 0,Y 175.344,Z 600.172,A -85,B 0,C 180,E1 -23339.402,E2 -23339.402} C_VEL
LIN {X 0,Y 179.493,Z 592.069,A -85,B 0,C 180,E1 -23342.569,E2 -23342.569} C_VEL
LIN {X 0,Y 184.179,Z 582.299,A -85,B 0,C 180,E1 -23345.582,E2 -23345.582} C_VEL
LIN {X 0,Y 188.89,Z 571.436,A -85,B 0,C 180,E1 -23348.208,E2 -23348.208} C_VEL
LIN {X 0,Y 190.604,Z 566.515,A -85,B 0,C 180,E1 -23349.256,E2 -23349.256} C_VEL
LIN {X 0,Y 191.192,Z 555.781,A -85,B 0,C 180,E1 -23351.965,E2 -23351.965} C_VEL
LIN {X 0,Y 190.819,Z 545.624,A -85,B 0,C 180,E1 -23354.405,E2 -23354.405} C_VEL
LIN {X 0,Y 189.471,Z 534.452,A -85,B 0,C 180,E1 -23357.033,E2 -23357.033} C_VEL
LIN {X 0,Y 188.236,Z 528.858,A -85,B 0,C 180,E1 -23358.42,E2 -23358.42} C_VEL
LIN {X 0,Y 184.914,Z 520.656,A -85,B 0,C 180,E1 -23360.9,E2 -23360.9} C_VEL
LIN {X 0,Y 181.373,Z 513.468,A -85,B 0,C 180,E1 -23363.314,E2 -23363.314} C_VEL
LIN {X 0,Y 178.849,Z 508.938,A -85,B 0,C 180,E1 -23364.981,E2 -23364.981} C_VEL
LIN {X 0,Y 176.066,Z 504.254,A -85,B 0,C 180,E1 -23366.842,E2 -23366.842} C_VEL
LIN {X 0,Y 173.359,Z 500.333,A -85,B 0,C 180,E1 -23368.621,E2 -23368.621} C_VEL
LIN {X 0,Y 172.525,Z 498.928,A -85,B 0,C 180,E1 -23369.219,E2 -23369.219} C_VEL
LIN {X 0,Y 169.677,Z 495.678,A -85,B 0,C 180,E1 -23371.169,E2 -23371.169} C_VEL
LIN {X 0,Y 168.391,Z 493.066,A -85,B 0,C 180,E1 -23372.287,E2 -23372.287} C_VEL
LIN {X 0,Y 167.655,Z 489.662,A -85,B 0,C 180,E1 -23377.835,E2 -23377.835} C_VEL
LIN {X 0,Y 167.081,Z 487.032,A -85,B 0,C 180,E1 -23382.876,E2 -23382.876} C_VEL
LIN {X 0,Y 166.622,Z 484.985,A -85,B 0,C 180,E1 -23387.825,E2 -23387.825} C_VEL
LIN {X 0,Y 166.618,Z 484.131,A -85,B 0,C 180,E1 -23390.286,E2 -23390.286} C_VEL
LIN {X 0,Y 166.231,Z 483.127,A -85,B 0,C 180,E1 -23395.149,E2 -23395.149} C_VEL
LIN {X 0,Y 166.412,Z 482.235,A -85,B 0,C 180,E1 -23400,E2 -23400} C_VEL
LIN {X 0,Y 166.046,Z 482.593,A -85,B 0,C 180,E1 -23404.856,E2 -23404.856} C_VEL
LIN {X 0,Y 166.356,Z 483.275,A -85,B 0,C 180,E1 -23409.729,E2 -23409.729} C_VEL
LIN {X 0,Y 166.716,Z 484.682,A -85,B 0,C 180,E1 -23414.651,E2 -23414.651} C_VEL
LIN {X 0,Y 167.324,Z 486.918,A -85,B 0,C 180,E1 -23419.634,E2 -23419.634} C_VEL
LIN {X 0,Y 168.394,Z 489.924,A -85,B 0,C 180,E1 -23424.668,E2 -23424.668} C_VEL
LIN {X 0,Y 169.619,Z 492.995,A -85,B 0,C 180,E1 -23428.745,E2 -23428.745} C_VEL
LIN {X 0,Y 172.396,Z 497.101,A -85,B 0,C 180,E1 -23430.721,E2 -23430.721} C_VEL
LIN {X 0,Y 174.344,Z 499.229,A -85,B 0,C 180,E1 -23431.953,E2 -23431.953} C_VEL
LIN {X 0,Y 177.483,Z 503.706,A -85,B 0,C 180,E1 -23433.939,E2 -23433.939} C_VEL
LIN {X 0,Y 181.877,Z 510.279,A -85,B 0,C 180,E1 -23436.588,E2 -23436.588} C_VEL
LIN {X 0,Y 184.522,Z 515.222,A -85,B 0,C 180,E1 -23438.237,E2 -23438.237} C_VEL
LIN {X 0,Y 188.95,Z 525.463,A -85,B 0,C 180,E1 -23441.227,E2 -23441.227} C_VEL
LIN {X 0,Y 192.739,Z 536.936,A -85,B 0,C 180,E1 -23444.296,E2 -23444.296} C_VEL
LIN {X 0,Y 193.109,Z 545.061,A -85,B 0,C 180,E1 -23445.903,E2 -23445.903} C_VEL
LIN {X 0,Y 192.366,Z 556.239,A -85,B 0,C 180,E1 -23448.112,E2 -23448.112} C_VEL
LIN {X 0,Y 191.031,Z 566.076,A -85,B 0,C 180,E1 -23450.27,E2 -23450.27} C_VEL
LIN {X 0,Y 186.804,Z 577.218,A -85,B 0,C 180,E1 -23452.578,E2 -23452.578} C_VEL
LIN {X 0,Y 182.114,Z 587.774,A -85,B 0,C 180,E1 -23455.308,E2 -23455.308} C_VEL
LIN {X 0,Y 177.554,Z 597.07,A -85,B 0,C 180,E1 -23458.371,E2 -23458.371} C_VEL
LIN {X 0,Y 173.564,Z 604.781,A -85,B 0,C 180,E1 -23461.593,E2 -23461.593} C_VEL
LIN {X 0,Y 169.651,Z 612.136,A -85,B 0,C 180,E1 -23465.531,E2 -23465.531} C_VEL
LIN {X 0,Y 166.299,Z 618.721,A -85,B 0,C 180,E1 -23470.243,E2 -23470.243} C_VEL
LIN {X 0,Y 163.757,Z 623.654,A -85,B 0,C 180,E1 -23475.081,E2 -23475.081} C_VEL
LIN {X 0,Y 162.378,Z 627.082,A -85,B 0,C 180,E1 -23480.034,E2 -23480.034} C_VEL
LIN {X 0,Y 161.8,Z 629.107,A -85,B 0,C 180,E1 -23485.019,E2 -23485.019} C_VEL
LIN {X 0,Y 161.821,Z 629.773,A -85,B 0,C 180,E1 -23490.003,E2 -23490.003} C_VEL
LIN {X 0,Y 161.801,Z 629.081,A -85,B 0,C 180,E1 -23494.987,E2 -23494.987} C_VEL
LIN {X 0,Y 162.38,Z 627.033,A -85,B 0,C 180,E1 -23499.973,E2 -23499.973} C_VEL
LIN {X 0,Y 163.611,Z 623.881,A -85,B 0,C 180,E1 -23504.543,E2 -23504.543} C_VEL
LIN {X 0,Y 163.472,Z 622.817,A -85,B 0,C 180,E1 -23505.888,E2 -23505.888} C_VEL
LIN {X 0,Y 161.668,Z 620.966,A -85,B 0,C 180,E1 -23508.086,E2 -23508.086} C_VEL
LIN {X 0,Y 160.079,Z 618.867,A -85,B 0,C 180,E1 -23510.301,E2 -23510.301} C_VEL
LIN {X 0,Y 160.279,Z 617.385,A -85,B 0,C 180,E1 -23511.625,E2 -23511.625} C_VEL
LIN {X 0,Y 162.66,Z 613.47,A -85,B 0,C 180,E1 -23514.529,E2 -23514.529} C_VEL
LIN {X 0,Y 168.86,Z 612.883,A -85,B 0,C 180,E1 -23519.966,E2 -23519.966} C_VEL
LIN {X 0,Y 175.467,Z 611.405,A -85,B 0,C 180,E1 -23524.11,E2 -23524.11} C_VEL
LIN {X 0,Y 183.205,Z 609.08,A -85,B 0,C 180,E1 -23527.867,E2 -23527.867} C_VEL
LIN {X 0,Y 191.975,Z 605.906,A -85,B 0,C 180,E1 -23531.224,E2 -23531.224} C_VEL
LIN {X 0,Y 204.255,Z 600.577,A -85,B 0,C 180,E1 -23534.862,E2 -23534.862} C_VEL
LIN {X 0,Y 212.24,Z 596.645,A -85,B 0,C 180,E1 -23536.763,E2 -23536.763} C_VEL
LIN {X 0,Y 212.25,Z 596.472,A -85,B 0,C 180,E1 -23537.654,E2 -23537.654} C_VEL
LIN {X 0,Y 200.229,Z 601.062,A -85,B 0,C 180,E1 -23540.817,E2 -23540.817} C_VEL
LIN {X 0,Y 190.794,Z 603.839,A -85,B 0,C 180,E1 -23543.888,E2 -23543.888} C_VEL
LIN {X 0,Y 182.274,Z 605.562,A -85,B 0,C 180,E1 -23547.33,E2 -23547.33} C_VEL
LIN {X 0,Y 174.804,Z 606.231,A -85,B 0,C 180,E1 -23551.154,E2 -23551.154} C_VEL
LIN {X 0,Y 168.419,Z 605.848,A -85,B 0,C 180,E1 -23555.336,E2 -23555.336} C_VEL
LIN {X 0,Y 163.337,Z 604.37,A -85,B 0,C 180,E1 -23559.866,E2 -23559.866} C_VEL
LIN {X 0,Y 159.549,Z 601.782,A -85,B 0,C 180,E1 -23564.675,E2 -23564.675} C_VEL
LIN {X 0,Y 156.939,Z 598.014,A -85,B 0,C 180,E1 -23569.681,E2 -23569.681} C_VEL
LIN {X 0,Y 155.749,Z 592.956,A -85,B 0,C 180,E1 -23574.822,E2 -23574.822} C_VEL
LIN {X 0,Y 155.473,Z 588.209,A -85,B 0,C 180,E1 -23578.705,E2 -23578.705} C_VEL
LIN {X 0,Y 155.495,Z 581.351,A -85,B 0,C 180,E1 -23583.239,E2 -23583.239} C_VEL
LIN {X 0,Y 155.901,Z 572.895,A -85,B 0,C 180,E1 -23587.773,E2 -23587.773} C_VEL
LIN {X 0,Y 156.734,Z 564.126,A -85,B 0,C 180,E1 -23591.641,E2 -23591.641} C_VEL
LIN {X 0,Y 158.036,Z 553.459,A -85,B 0,C 180,E1 -23595.476,E2 -23595.476} C_VEL
LIN {X 0,Y 159.739,Z 541.813,A -85,B 0,C 180,E1 -23598.934,E2 -23598.934} C_VEL
LIN {X 0,Y 161.661,Z 528.959,A -85,B 0,C 180,E1 -23602.022,E2 -23602.022} C_VEL
LIN {X 0,Y 159.983,Z 516.385,A -85,B 0,C 180,E1 -23604.528,E2 -23604.528} C_VEL
LIN {X 0,Y 159.677,Z 514.41,A -85,B 0,C 180,E1 -23604.912,E2 -23604.912} C_VEL
LIN {X 0,Y 160.113,Z 515.433,A -85,B 0,C 180,E1 -23605.461,E2 -23605.461} C_VEL
LIN {X 0,Y 161.005,Z 515.626,A -85,B 0,C 180,E1 -23606.159,E2 -23606.159} C_VEL
LIN {X 0,Y 162.508,Z 514.465,A -85,B 0,C 180,E1 -23606.994,E2 -23606.994} C_VEL
LIN {X 0,Y 164.445,Z 511.821,A -85,B 0,C 180,E1 -23607.801,E2 -23607.801} C_VEL
LIN {X 0,Y 165.604,Z 509.803,A -85,B 0,C 180,E1 -23608.242,E2 -23608.242} C_VEL
LIN {X 0,Y 167.685,Z 508.588,A -85,B 0,C 180,E1 -23609.367,E2 -23609.367} C_VEL
LIN {X 0,Y 169.084,Z 507.368,A -85,B 0,C 180,E1 -23610.032,E2 -23610.032} C_VEL
LIN {X 0,Y 172.805,Z 511.351,A -85,B 0,C 180,E1 -23612.608,E2 -23612.608} C_VEL
LIN {X 0,Y 176.562,Z 516.879,A -85,B 0,C 180,E1 -23615.252,E2 -23615.252} C_VEL
LIN {X 0,Y 179.358,Z 522.685,A -85,B 0,C 180,E1 -23617.399,E2 -23617.399} C_VEL
LIN {X 0,Y 182.881,Z 531.602,A -85,B 0,C 180,E1 -23620.347,E2 -23620.347} C_VEL
LIN {X 0,Y 184.099,Z 536.731,A -85,B 0,C 180,E1 -23621.767,E2 -23621.767} C_VEL
LIN {X 0,Y 185.218,Z 547.965,A -85,B 0,C 180,E1 -23624.584,E2 -23624.584} C_VEL
LIN {X 0,Y 185.271,Z 558.642,A -85,B 0,C 180,E1 -23627.305,E2 -23627.305} C_VEL
LIN {X 0,Y 184.407,Z 568.484,A -85,B 0,C 180,E1 -23629.93,E2 -23629.93} C_VEL
LIN {X 0,Y 179.399,Z 580.037,A -85,B 0,C 180,E1 -23632.608,E2 -23632.608} C_VEL
LIN {X 0,Y 174.382,Z 590.253,A -85,B 0,C 180,E1 -23635.648,E2 -23635.648} C_VEL
LIN {X 0,Y 169.966,Z 598.676,A -85,B 0,C 180,E1 -23638.874,E2 -23638.874} C_VEL
LIN {X 0,Y 165.319,Z 606.81,A -85,B 0,C 180,E1 -23642.871,E2 -23642.871} C_VEL
LIN {X 0,Y 161.813,Z 613.169,A -85,B 0,C 180,E1 -23646.987,E2 -23646.987} C_VEL
LIN {X 0,Y 159.248,Z 617.638,A -85,B 0,C 180,E1 -23650.668,E2 -23650.668} C_VEL
LIN {X 0,Y 157.281,Z 621.144,A -85,B 0,C 180,E1 -23654.445,E2 -23654.445} C_VEL
LIN {X 0,Y 155.598,Z 624.564,A -85,B 0,C 180,E1 -23659.588,E2 -23659.588} C_VEL
LIN {X 0,Y 154.772,Z 626.596,A -85,B 0,C 180,E1 -23664.786,E2 -23664.786} C_VEL
LIN {X 0,Y 154.705,Z 627.289,A -85,B 0,C 180,E1 -23669.997,E2 -23669.997} C_VEL
LIN {X 0,Y 154.77,Z 626.649,A -85,B 0,C 180,E1 -23675.207,E2 -23675.207} C_VEL
LIN {X 0,Y 155.569,Z 624.663,A -85,B 0,C 180,E1 -23680.407,E2 -23680.407} C_VEL
LIN {X 0,Y 157.229,Z 621.286,A -85,B 0,C 180,E1 -23685.553,E2 -23685.553} C_VEL
LIN {X 0,Y 159.181,Z 617.813,A -85,B 0,C 180,E1 -23689.334,E2 -23689.334} C_VEL
LIN {X 0,Y 161.756,Z 613.377,A -85,B 0,C 180,E1 -23693.015,E2 -23693.015} C_VEL
LIN {X 0,Y 165.339,Z 606.973,A -85,B 0,C 180,E1 -23697.186,E2 -23697.186} C_VEL
LIN {X 0,Y 169.887,Z 599.006,A -85,B 0,C 180,E1 -23701.135,E2 -23701.135} C_VEL
LIN {X 0,Y 174.295,Z 590.651,A -85,B 0,C 180,E1 -23704.365,E2 -23704.365} C_VEL
LIN {X 0,Y 179.345,Z 580.537,A -85,B 0,C 180,E1 -23707.398,E2 -23707.398} C_VEL
LIN {X 0,Y 184.349,Z 568.988,A -85,B 0,C 180,E1 -23710.107,E2 -23710.107} C_VEL
LIN {X 0,Y 185.246,Z 560.707,A -85,B 0,C 180,E1 -23712.326,E2 -23712.326} C_VEL
LIN {X 0,Y 185.421,Z 551.38,A -85,B 0,C 180,E1 -23714.71,E2 -23714.71} C_VEL
LIN {X 0,Y 184.602,Z 539.826,A -85,B 0,C 180,E1 -23717.605,E2 -23717.605} C_VEL
LIN {X 0,Y 183.441,Z 533.095,A -85,B 0,C 180,E1 -23719.36,E2 -23719.36} C_VEL
LIN {X 0,Y 180.293,Z 524.563,A -85,B 0,C 180,E1 -23722.124,E2 -23722.124} C_VEL
LIN {X 0,Y 177.17,Z 517.96,A -85,B 0,C 180,E1 -23724.539,E2 -23724.539} C_VEL
LIN {X 0,Y 174.954,Z 513.76,A -85,B 0,C 180,E1 -23726.192,E2 -23726.192} C_VEL
LIN {X 0,Y 172.833,Z 509.912,A -85,B 0,C 180,E1 -23727.809,E2 -23727.809} C_VEL
LIN {X 0,Y 170.245,Z 505.644,A -85,B 0,C 180,E1 -23729.793,E2 -23729.793} C_VEL
LIN {X 0,Y 166.944,Z 501.289,A -85,B 0,C 180,E1 -23732.32,E2 -23732.32} C_VEL
LIN {X 0,Y 165.727,Z 499.139,A -85,B 0,C 180,E1 -23733.389,E2 -23733.389} C_VEL
LIN {X 0,Y 162.67,Z 495.616,A -85,B 0,C 180,E1 -23736.018,E2 -23736.018} C_VEL
LIN {X 0,Y 161.365,Z 493.075,A -85,B 0,C 180,E1 -23737.429,E2 -23737.429} C_VEL
LIN {X 0,Y 160.858,Z 490.698,A -85,B 0,C 180,E1 -23742.191,E2 -23742.191} C_VEL
LIN {X 0,Y 160.483,Z 488.721,A -85,B 0,C 180,E1 -23747.352,E2 -23747.352} C_VEL
LIN {X 0,Y 160.465,Z 487.861,A -85,B 0,C 180,E1 -23749.91,E2 -23749.91} C_VEL
LIN {X 0,Y 160.309,Z 487.174,A -85,B 0,C 180,E1 -23752.442,E2 -23752.442} C_VEL
LIN {X 0,Y 160.354,Z 485.949,A -85,B 0,C 180,E1 -23760,E2 -23760} C_VEL
LIN {X 0,Y 160.064,Z 486.418,A -85,B 0,C 180,E1 -23765.038,E2 -23765.038} C_VEL
LIN {X 0,Y 160.381,Z 487.2,A -85,B 0,C 180,E1 -23770.095,E2 -23770.095} C_VEL
LIN {X 0,Y 160.79,Z 488.784,A -85,B 0,C 180,E1 -23775.204,E2 -23775.204} C_VEL
LIN {X 0,Y 161.443,Z 491.14,A -85,B 0,C 180,E1 -23780.381,E2 -23780.381} C_VEL
LIN {X 0,Y 162.135,Z 493.002,A -85,B 0,C 180,E1 -23783.451,E2 -23783.451} C_VEL
LIN {X 0,Y 165.178,Z 497.203,A -85,B 0,C 180,E1 -23786.195,E2 -23786.195} C_VEL
LIN {X 0,Y 167.472,Z 499.554,A -85,B 0,C 180,E1 -23787.973,E2 -23787.973} C_VEL
LIN {X 0,Y 170.391,Z 503.778,A -85,B 0,C 180,E1 -23790.21,E2 -23790.21} C_VEL
LIN {X 0,Y 171.788,Z 505.586,A -85,B 0,C 180,E1 -23791.183,E2 -23791.183} C_VEL
LIN {X 0,Y 175.953,Z 511.88,A -85,B 0,C 180,E1 -23794.086,E2 -23794.086} C_VEL
LIN {X 0,Y 178.885,Z 516.895,A -85,B 0,C 180,E1 -23796.108,E2 -23796.108} C_VEL
LIN {X 0,Y 181.762,Z 523.108,A -85,B 0,C 180,E1 -23798.218,E2 -23798.218} C_VEL
LIN {X 0,Y 185.683,Z 533.97,A -85,B 0,C 180,E1 -23801.48,E2 -23801.48} C_VEL
LIN {X 0,Y 187.537,Z 540.655,A -85,B 0,C 180,E1 -23803.356,E2 -23803.356} C_VEL
LIN {X 0,Y 187.489,Z 548.927,A -85,B 0,C 180,E1 -23805.067,E2 -23805.067} C_VEL
LIN {X 0,Y 186.205,Z 560.774,A -85,B 0,C 180,E1 -23807.576,E2 -23807.576} C_VEL
LIN {X 0,Y 185.172,Z 567.316,A -85,B 0,C 180,E1 -23809.107,E2 -23809.107} C_VEL
LIN {X 0,Y 180.631,Z 578.459,A -85,B 0,C 180,E1 -23811.503,E2 -23811.503} C_VEL
LIN {X 0,Y 175.462,Z 589.372,A -85,B 0,C 180,E1 -23814.498,E2 -23814.498} C_VEL
LIN {X 0,Y 170.783,Z 598.371,A -85,B 0,C 180,E1 -23817.662,E2 -23817.662} C_VEL
LIN {X 0,Y 166.034,Z 606.965,A -85,B 0,C 180,E1 -23821.566,E2 -23821.566} C_VEL
LIN {X 0,Y 162.034,Z 614.121,A -85,B 0,C 180,E1 -23825.848,E2 -23825.848} C_VEL
LIN {X 0,Y 158.82,Z 620.082,A -85,B 0,C 180,E1 -23830.62,E2 -23830.62} C_VEL
LIN {X 0,Y 156.862,Z 623.599,A -85,B 0,C 180,E1 -23834.409,E2 -23834.409} C_VEL
LIN {X 0,Y 155.347,Z 627.027,A -85,B 0,C 180,E1 -23839.578,E2 -23839.578} C_VEL
LIN {X 0,Y 154.716,Z 629.052,A -85,B 0,C 180,E1 -23844.791,E2 -23844.791} C_VEL
LIN {X 0,Y 154.744,Z 629.717,A -85,B 0,C 180,E1 -23850.003,E2 -23850.003} C_VEL
LIN {X 0,Y 154.718,Z 629.025,A -85,B 0,C 180,E1 -23855.216,E2 -23855.216} C_VEL
LIN {X 0,Y 155.349,Z 626.977,A -85,B 0,C 180,E1 -23860.429,E2 -23860.429} C_VEL
LIN {X 0,Y 156.86,Z 623.528,A -85,B 0,C 180,E1 -23865.598,E2 -23865.598} C_VEL
LIN {X 0,Y 159.607,Z 618.578,A -85,B 0,C 180,E1 -23870.629,E2 -23870.629} C_VEL
LIN {X 0,Y 160.279,Z 617.385,A -85,B 0,C 180,E1 -23871.625,E2 -23871.625} C_VEL
LIN {X 0,Y 160.578,Z 615.948,A -85,B 0,C 180,E1 -23872.963,E2 -23872.963} C_VEL
LIN {X 0,Y 159.601,Z 614.146,A -85,B 0,C 180,E1 -23875.286,E2 -23875.286} C_VEL
LIN {X 0,Y 159.031,Z 613.075,A -85,B 0,C 180,E1 -23877.678,E2 -23877.678} C_VEL
LIN {X 0,Y 159.933,Z 612.793,A -85,B 0,C 180,E1 -23879.069,E2 -23879.069} C_VEL
LIN {X 0,Y 166.043,Z 612.148,A -85,B 0,C 180,E1 -23883.387,E2 -23883.387} C_VEL
LIN {X 0,Y 173.487,Z 610.601,A -85,B 0,C 180,E1 -23887.423,E2 -23887.423} C_VEL
LIN {X 0,Y 182.051,Z 608.249,A -85,B 0,C 180,E1 -23891.02,E2 -23891.02} C_VEL
LIN {X 0,Y 191.641,Z 605.035,A -85,B 0,C 180,E1 -23894.173,E2 -23894.173} C_VEL
LIN {X 0,Y 202.064,Z 600.908,A -85,B 0,C 180,E1 -23896.923,E2 -23896.923} C_VEL
LIN {X 0,Y 202.61,Z 600.598,A -85,B 0,C 180,E1 -23897.498,E2 -23897.498} C_VEL
LIN {X 0,Y 194.926,Z 602.95,A -85,B 0,C 180,E1 -23899.535,E2 -23899.535} C_VEL
LIN {X 0,Y 185.215,Z 605.257,A -85,B 0,C 180,E1 -23902.618,E2 -23902.618} C_VEL
LIN {X 0,Y 176.402,Z 606.544,A -85,B 0,C 180,E1 -23906.098,E2 -23906.098} C_VEL
LIN {X 0,Y 168.664,Z 606.819,A -85,B 0,C 180,E1 -23909.999,E2 -23909.999} C_VEL
LIN {X 0,Y 162,Z 606.055,A -85,B 0,C 180,E1 -23914.29,E2 -23914.29} C_VEL
LIN {X 0,Y 156.699,Z 604.224,A -85,B 0,C 180,E1 -23918.973,E2 -23918.973} C_VEL
